LIN {X 0,Y 249.453,Z 553.415,A -85,B 0,C 180,E1 -18983.532,E2 -18983.532} C_VEL
LIN {X 0,Y 249.673,Z 553.384,A -85,B 0,C 180,E1 -18988.389,E2 -18988.389} C_VEL
LIN {X 0,Y 249.674,Z 553.383,A -85,B 0,C 180,E1 -18991.615,E2 -18991.615} C_VEL
LIN {X 0,Y 249.457,Z 553.406,A -85,B 0,C 180,E1 -18996.473,E2 -18996.473} C_VEL
LIN {X 0,Y 249.387,Z 553.419,A -85,B 0,C 180,E1 -18999.737,E2 -18999.737} C_VEL
LIN {X 0,Y 249.205,Z 553.438,A -85,B 0,C 180,E1 -19004.706,E2 -19004.706} C_VEL
LIN {X 0,Y 249.14,Z 553.449,A -85,B 0,C 180,E1 -19008.08,E2 -19008.08} C_VEL
LIN {X 0,Y 249.088,Z 553.442,A -85,B 0,C 180,E1 -19011.52,E2 -19011.52} C_VEL
LIN {X 0,Y 249.131,Z 553.45,A -85,B 0,C 180,E1 -19015.484,E2 -19015.484} C_VEL
LIN {X 0,Y 249.074,Z 553.461,A -85,B 0,C 180,E1 -19018.991,E2 -19018.991} C_VEL
LIN {X 0,Y 249.032,Z 553.458,A -85,B 0,C 180,E1 -19022.428,E2 -19022.428} C_VEL
LIN {X 0,Y 249.032,Z 553.463,A -85,B 0,C 180,E1 -19026.348,E2 -19026.348} C_VEL
LIN {X 0,Y 249.009,Z 553.46,A -85,B 0,C 180,E1 -19030.48,E2 -19030.48} C_VEL
LIN {X 0,Y 249.011,Z 553.466,A -85,B 0,C 180,E1 -19034.88,E2 -19034.88} C_VEL
LIN {X 0,Y 249.022,Z 553.465,A -85,B 0,C 180,E1 -19037.365,E2 -19037.365} C_VEL
LIN {X 0,Y 249.048,Z 553.457,A -85,B 0,C 180,E1 -19042.202,E2 -19042.202} C_VEL
LIN {X 0,Y 249.049,Z 553.463,A -85,B 0,C 180,E1 -19045.641,E2 -19045.641} C_VEL
LIN {X 0,Y 249.058,Z 553.456,A -85,B 0,C 180,E1 -19049.475,E2 -19049.475} C_VEL
LIN {X 0,Y 249.076,Z 553.452,A -85,B 0,C 180,E1 -19053.164,E2 -19053.164} C_VEL
LIN {X 0,Y 249.067,Z 553.458,A -85,B 0,C 180,E1 -19056.732,E2 -19056.732} C_VEL
LIN {X 0,Y 249.092,Z 553.451,A -85,B 0,C 180,E1 -19060.211,E2 -19060.211} C_VEL
LIN {X 0,Y 249.203,Z 553.435,A -85,B 0,C 180,E1 -19063.62,E2 -19063.62} C_VEL
LIN {X 0,Y 249.251,Z 553.435,A -85,B 0,C 180,E1 -19068.617,E2 -19068.617} C_VEL
LIN {X 0,Y 249.463,Z 553.405,A -85,B 0,C 180,E1 -19071.903,E2 -19071.903} C_VEL
LIN {X 0,Y 249.303,Z 553.423,A -85,B 0,C 180,E1 -19075.149,E2 -19075.149} C_VEL
LIN {X 0,Y 249.683,Z 553.382,A -85,B 0,C 180,E1 -19078.388,E2 -19078.388} C_VEL
LIN {X 0,Y 249.684,Z 553.383,A -85,B 0,C 180,E1 -19081.614,E2 -19081.614} C_VEL
LIN {X 0,Y 249.47,Z 553.408,A -85,B 0,C 180,E1 -19086.471,E2 -19086.471} C_VEL
LIN {X 0,Y 249.434,Z 553.416,A -85,B 0,C 180,E1 -19089.734,E2 -19089.734} C_VEL
LIN {X 0,Y 249.224,Z 553.432,A -85,B 0,C 180,E1 -19092.092,E2 -19092.092} C_VEL
LIN {X 0,Y 248.533,Z 553.52,A -85,B 0,C 180,E1 -19093.442,E2 -19093.442} C_VEL
LIN {X 0,Y 245.654,Z 553.884,A -85,B 0,C 180,E1 -19095.642,E2 -19095.642} C_VEL
LIN {X 0,Y 243.205,Z 554.19,A -85,B 0,C 180,E1 -19097.434,E2 -19097.434} C_VEL
LIN {X 0,Y 242.137,Z 554.321,A -85,B 0,C 180,E1 -19098.824,E2 -19098.824} C_VEL
LIN {X 0,Y 242.04,Z 554.328,A -85,B 0,C 180,E1 -19099.296,E2 -19099.296} C_VEL
LIN {X 0,Y 242.05,Z 554.315,A -85,B 0,C 180,E1 -19103.986,E2 -19103.986} C_VEL
LIN {X 0,Y 242.01,Z 554.334,A -85,B 0,C 180,E1 -19107.688,E2 -19107.688} C_VEL
LIN {X 0,Y 241.983,Z 554.34,A -85,B 0,C 180,E1 -19111.52,E2 -19111.52} C_VEL
LIN {X 0,Y 242.015,Z 554.338,A -85,B 0,C 180,E1 -19115.596,E2 -19115.596} C_VEL
LIN {X 0,Y 241.965,Z 554.344,A -85,B 0,C 180,E1 -19119.718,E2 -19119.718} C_VEL
LIN {X 0,Y 241.935,Z 554.349,A -85,B 0,C 180,E1 -19124.202,E2 -19124.202} C_VEL
LIN {X 0,Y 241.947,Z 554.347,A -85,B 0,C 180,E1 -19128.077,E2 -19128.077} C_VEL
LIN {X 0,Y 242.02,Z 554.338,A -85,B 0,C 180,E1 -19132.421,E2 -19132.421} C_VEL
LIN {X 0,Y 242.101,Z 554.421,A -85,B 0,C 180,E1 -19133.371,E2 -19133.371} C_VEL
LIN {X 0,Y 244.113,Z 564.051,A -85,B 0,C 180,E1 -19137.327,E2 -19137.327} C_VEL
LIN {X 0,Y 245.054,Z 568.388,A -85,B 0,C 180,E1 -19138.956,E2 -19138.956} C_VEL
LIN {X 0,Y 252.11,Z 587.582,A -85,B 0,C 180,E1 -19140.375,E2 -19140.375} C_VEL
LIN {X 0,Y 256.177,Z 617.752,A -85,B 0,C 180,E1 -19141.803,E2 -19141.803} C_VEL
LIN {X 0,Y 253.863,Z 677.446,A -85,B 0,C 180,E1 -19143.657,E2 -19143.657} C_VEL
LIN {X 0,Y 252.711,Z 691.266,A -85,B 0,C 180,E1 -19144.408,E2 -19144.408} C_VEL
LIN {X 0,Y 251.292,Z 703.771,A -85,B 0,C 180,E1 -19145.414,E2 -19145.414} C_VEL
LIN {X 0,Y 249.549,Z 716.207,A -85,B 0,C 180,E1 -19146.777,E2 -19146.777} C_VEL
LIN {X 0,Y 247.692,Z 727.365,A -85,B 0,C 180,E1 -19148.352,E2 -19148.352} C_VEL
LIN {X 0,Y 245.909,Z 737.764,A -85,B 0,C 180,E1 -19150.23,E2 -19150.23} C_VEL
LIN {X 0,Y 244.312,Z 747.422,A -85,B 0,C 180,E1 -19152.417,E2 -19152.417} C_VEL
LIN {X 0,Y 242.903,Z 754.812,A -85,B 0,C 180,E1 -19154.474,E2 -19154.474} C_VEL
LIN {X 0,Y 241.522,Z 762.054,A -85,B 0,C 180,E1 -19156.964,E2 -19156.964} C_VEL
LIN {X 0,Y 240.812,Z 766.949,A -85,B 0,C 180,E1 -19159.062,E2 -19159.062} C_VEL
LIN {X 0,Y 240.212,Z 771.663,A -85,B 0,C 180,E1 -19161.586,E2 -19161.586} C_VEL
LIN {X 0,Y 239.907,Z 775.221,A -85,B 0,C 180,E1 -19164.113,E2 -19164.113} C_VEL
LIN {X 0,Y 239.806,Z 777.727,A -85,B 0,C 180,E1 -19166.637,E2 -19166.637} C_VEL
LIN {X 0,Y 239.866,Z 778.859,A -85,B 0,C 180,E1 -19168.319,E2 -19168.319} C_VEL
LIN {X 0,Y 239.915,Z 779.546,A -85,B 0,C 180,E1 -19169.998,E2 -19169.998} C_VEL
LIN {X 0,Y 239.833,Z 779.83,A -85,B 0,C 180,E1 -19171.677,E2 -19171.677} C_VEL
LIN {X 0,Y 239.793,Z 779.295,A -85,B 0,C 180,E1 -19174.791,E2 -19174.791} C_VEL
LIN {X 0,Y 239.954,Z 778.232,A -85,B 0,C 180,E1 -19176.726,E2 -19176.726} C_VEL
LIN {X 0,Y 240.672,Z 775.128,A -85,B 0,C 180,E1 -19180.088,E2 -19180.088} C_VEL
LIN {X 0,Y 241.623,Z 771.637,A -85,B 0,C 180,E1 -19182.598,E2 -19182.598} C_VEL
LIN {X 0,Y 242.985,Z 767.08,A -85,B 0,C 180,E1 -19185.086,E2 -19185.086} C_VEL
LIN {X 0,Y 245.294,Z 760.216,A -85,B 0,C 180,E1 -19187.936,E2 -19187.936} C_VEL
LIN {X 0,Y 247.599,Z 752.325,A -85,B 0,C 180,E1 -19190.495,E2 -19190.495} C_VEL
LIN {X 0,Y 250.22,Z 743.627,A -85,B 0,C 180,E1 -19192.716,E2 -19192.716} C_VEL
LIN {X 0,Y 253.211,Z 733.103,A -85,B 0,C 180,E1 -19194.819,E2 -19194.819} C_VEL
LIN {X 0,Y 255.815,Z 722.508,A -85,B 0,C 180,E1 -19196.512,E2 -19196.512} C_VEL
LIN {X 0,Y 258.523,Z 710.623,A -85,B 0,C 180,E1 -19197.963,E2 -19197.963} C_VEL
LIN {X 0,Y 260.759,Z 698.126,A -85,B 0,C 180,E1 -19199.129,E2 -19199.129} C_VEL
LIN {X 0,Y 262.607,Z 685.023,A -85,B 0,C 180,E1 -19200.005,E2 -19200.005} C_VEL
LIN {X 0,Y 263.954,Z 670.854,A -85,B 0,C 180,E1 -19200.603,E2 -19200.603} C_VEL
LIN {X 0,Y 266.576,Z 619.411,A -85,B 0,C 180,E1 -19202.173,E2 -19202.173} C_VEL
LIN {X 0,Y 264.465,Z 603.384,A -85,B 0,C 180,E1 -19203.2,E2 -19203.2} C_VEL
LIN {X 0,Y 260.104,Z 593.001,A -85,B 0,C 180,E1 -19204.48,E2 -19204.48} C_VEL
LIN {X 0,Y 253.772,Z 580.509,A -85,B 0,C 180,E1 -19206.375,E2 -19206.375} C_VEL
LIN {X 0,Y 250.696,Z 575.081,A -85,B 0,C 180,E1 -19207.34,E2 -19207.34} C_VEL
LIN {X 0,Y 247.979,Z 570.475,A -85,B 0,C 180,E1 -19208.225,E2 -19208.225} C_VEL
LIN {X 0,Y 245.387,Z 565.842,A -85,B 0,C 180,E1 -19209.17,E2 -19209.17} C_VEL
LIN {X 0,Y 243.644,Z 560.104,A -85,B 0,C 180,E1 -19212.645,E2 -19212.645} C_VEL
LIN {X 0,Y 241.944,Z 554.347,A -85,B 0,C 180,E1 -19216.7,E2 -19216.7} C_VEL
LIN {X 0,Y 241.975,Z 554.339,A -85,B 0,C 180,E1 -19220.284,E2 -19220.284} C_VEL
LIN {X 0,Y 242.03,Z 554.338,A -85,B 0,C 180,E1 -19224.495,E2 -19224.495} C_VEL
LIN {X 0,Y 241.968,Z 554.338,A -85,B 0,C 180,E1 -19228.478,E2 -19228.478} C_VEL
LIN {X 0,Y 242,Z 554.332,A -85,B 0,C 180,E1 -19232.311,E2 -19232.311} C_VEL
LIN {X 0,Y 242.049,Z 554.325,A -85,B 0,C 180,E1 -19236.014,E2 -19236.014} C_VEL
LIN {X 0,Y 242.028,Z 554.328,A -85,B 0,C 180,E1 -19239.606,E2 -19239.606} C_VEL
LIN {X 0,Y 242.154,Z 554.315,A -85,B 0,C 180,E1 -19243.277,E2 -19243.277} C_VEL
LIN {X 0,Y 242.177,Z 554.308,A -85,B 0,C 180,E1 -19248.278,E2 -19248.278} C_VEL
LIN {X 0,Y 242.425,Z 554.278,A -85,B 0,C 180,E1 -19251.665,E2 -19251.665} C_VEL
LIN {X 0,Y 242.252,Z 554.301,A -85,B 0,C 180,E1 -19255.006,E2 -19255.006} C_VEL
LIN {X 0,Y 242.629,Z 554.255,A -85,B 0,C 180,E1 -19258.339,E2 -19258.339} C_VEL
LIN {X 0,Y 242.634,Z 554.256,A -85,B 0,C 180,E1 -19261.659,E2 -19261.659} C_VEL
LIN {X 0,Y 242.427,Z 554.334,A -85,B 0,C 180,E1 -19267.914,E2 -19267.914} C_VEL
LIN {X 0,Y 243.227,Z 557.795,A -85,B 0,C 180,E1 -19270.351,E2 -19270.351} C_VEL
LIN {X 0,Y 245.42,Z 561.512,A -85,B 0,C 180,E1 -19271.144,E2 -19271.144} C_VEL
LIN {X 0,Y 247.197,Z 563.941,A -85,B 0,C 180,E1 -19271.738,E2 -19271.738} C_VEL
LIN {X 0,Y 250.763,Z 569.544,A -85,B 0,C 180,E1 -19272.904,E2 -19272.904} C_VEL
LIN {X 0,Y 255.426,Z 577.254,A -85,B 0,C 180,E1 -19274.337,E2 -19274.337} C_VEL
LIN {X 0,Y 260.585,Z 586.905,A -85,B 0,C 180,E1 -19275.848,E2 -19275.848} C_VEL
LIN {X 0,Y 265.939,Z 598.808,A -85,B 0,C 180,E1 -19277.377,E2 -19277.377} C_VEL
LIN {X 0,Y 267.443,Z 602.427,A -85,B 0,C 180,E1 -19277.8,E2 -19277.8} C_VEL
LIN {X 0,Y 263.978,Z 664.442,A -85,B 0,C 180,E1 -19279.693,E2 -19279.693} C_VEL
LIN {X 0,Y 262.673,Z 677.208,A -85,B 0,C 180,E1 -19280.353,E2 -19280.353} C_VEL
LIN {X 0,Y 260.893,Z 690.002,A -85,B 0,C 180,E1 -19281.324,E2 -19281.324} C_VEL
LIN {X 0,Y 258.594,Z 702.502,A -85,B 0,C 180,E1 -19282.627,E2 -19282.627} C_VEL
LIN {X 0,Y 256.222,Z 713.303,A -85,B 0,C 180,E1 -19284.087,E2 -19284.087} C_VEL
LIN {X 0,Y 253.528,Z 724.026,A -85,B 0,C 180,E1 -19285.934,E2 -19285.934} C_VEL
LIN {X 0,Y 250.699,Z 733.84,A -85,B 0,C 180,E1 -19288.081,E2 -19288.081} C_VEL
LIN {X 0,Y 248.21,Z 741.845,A -85,B 0,C 180,E1 -19290.272,E2 -19290.272} C_VEL
LIN {X 0,Y 246.081,Z 748.371,A -85,B 0,C 180,E1 -19292.505,E2 -19292.505} C_VEL
LIN {X 0,Y 243.964,Z 754.493,A -85,B 0,C 180,E1 -19295.179,E2 -19295.179} C_VEL
LIN {X 0,Y 242.565,Z 758.575,A -85,B 0,C 180,E1 -19297.476,E2 -19297.476} C_VEL
LIN {X 0,Y 241.136,Z 762.726,A -85,B 0,C 180,E1 -19300.735,E2 -19300.735} C_VEL
LIN {X 0,Y 240.385,Z 764.662,A -85,B 0,C 180,E1 -19303.041,E2 -19303.041} C_VEL
LIN {X 0,Y 239.891,Z 765.829,A -85,B 0,C 180,E1 -19305.326,E2 -19305.326} C_VEL
LIN {X 0,Y 239.58,Z 766.222,A -85,B 0,C 180,E1 -19307.573,E2 -19307.573} C_VEL
LIN {X 0,Y 239.453,Z 765.906,A -85,B 0,C 180,E1 -19309.785,E2 -19309.785} C_VEL
LIN {X 0,Y 239.507,Z 764.641,A -85,B 0,C 180,E1 -19312.397,E2 -19312.397} C_VEL
LIN {X 0,Y 239.812,Z 762.222,A -85,B 0,C 180,E1 -19315.141,E2 -19315.141} C_VEL
LIN {X 0,Y 240.468,Z 758.038,A -85,B 0,C 180,E1 -19318.263,E2 -19318.263} C_VEL
LIN {X 0,Y 241.28,Z 753.121,A -85,B 0,C 180,E1 -19320.906,E2 -19320.906} C_VEL
LIN {X 0,Y 242.421,Z 746.61,A -85,B 0,C 180,E1 -19323.596,E2 -19323.596} C_VEL
LIN {X 0,Y 243.952,Z 738.534,A -85,B 0,C 180,E1 -19326.217,E2 -19326.217} C_VEL
LIN {X 0,Y 245.532,Z 730.166,A -85,B 0,C 180,E1 -19328.378,E2 -19328.378} C_VEL
LIN {X 0,Y 247.276,Z 719.954,A -85,B 0,C 180,E1 -19330.494,E2 -19330.494} C_VEL
LIN {X 0,Y 249.194,Z 708.613,A -85,B 0,C 180,E1 -19332.351,E2 -19332.351} C_VEL
LIN {X 0,Y 250.796,Z 696.998,A -85,B 0,C 180,E1 -19333.833,E2 -19333.833} C_VEL
LIN {X 0,Y 252.352,Z 684.2,A -85,B 0,C 180,E1 -19335.074,E2 -19335.074} C_VEL
LIN {X 0,Y 253.441,Z 671.386,A -85,B 0,C 180,E1 -19335.968,E2 -19335.968} C_VEL
LIN {X 0,Y 254.324,Z 657.187,A -85,B 0,C 180,E1 -19336.593,E2 -19336.593} C_VEL
LIN {X 0,Y 256.812,Z 593.445,A -85,B 0,C 180,E1 -19338.515,E2 -19338.515} C_VEL
LIN {X 0,Y 249.263,Z 572.337,A -85,B 0,C 180,E1 -19340.004,E2 -19340.004} C_VEL
LIN {X 0,Y 242.612,Z 555.291,A -85,B 0,C 180,E1 -19341.36,E2 -19341.36} C_VEL
LIN {X 0,Y 242.438,Z 554.287,A -85,B 0,C 180,E1 -19341.878,E2 -19341.878} C_VEL
LIN {X 0,Y 242.372,Z 554.299,A -85,B 0,C 180,E1 -19346.678,E2 -19346.678} C_VEL
LIN {X 0,Y 242.634,Z 554.261,A -85,B 0,C 180,E1 -19348.343,E2 -19348.343} C_VEL
LIN {X 0,Y 242.634,Z 554.259,A -85,B 0,C 180,E1 -19351.662,E2 -19351.662} C_VEL
LIN {X 0,Y 242.43,Z 554.282,A -85,B 0,C 180,E1 -19356.661,E2 -19356.661} C_VEL
LIN {X 0,Y 242.313,Z 554.3,A -85,B 0,C 180,E1 -19360.024,E2 -19360.024} C_VEL
LIN {X 0,Y 242.166,Z 554.318,A -85,B 0,C 180,E1 -19365.143,E2 -19365.143} C_VEL
LIN {X 0,Y 242.073,Z 554.33,A -85,B 0,C 180,E1 -19368.626,E2 -19368.626} C_VEL
LIN {X 0,Y 242.014,Z 554.32,A -85,B 0,C 180,E1 -19372.182,E2 -19372.182} C_VEL
LIN {X 0,Y 242.068,Z 554.329,A -85,B 0,C 180,E1 -19375.84,E2 -19375.84} C_VEL
LIN {X 0,Y 242.009,Z 554.339,A -85,B 0,C 180,E1 -19379.586,E2 -19379.586} C_VEL
LIN {X 0,Y 241.983,Z 554.342,A -85,B 0,C 180,E1 -19383.495,E2 -19383.495} C_VEL
LIN {X 0,Y 241.989,Z 554.341,A -85,B 0,C 180,E1 -19387.585,E2 -19387.585} C_VEL
LIN {X 0,Y 241.942,Z 554.343,A -85,B 0,C 180,E1 -19391.924,E2 -19391.924} C_VEL
LIN {X 0,Y 241.941,Z 554.346,A -85,B 0,C 180,E1 -19396.573,E2 -19396.573} C_VEL
LIN {X 0,Y 241.961,Z 554.333,A -85,B 0,C 180,E1 -19400.283,E2 -19400.283} C_VEL
LIN {X 0,Y 241.992,Z 554.339,A -85,B 0,C 180,E1 -19404.491,E2 -19404.491} C_VEL
LIN {X 0,Y 241.98,Z 554.338,A -85,B 0,C 180,E1 -19408.482,E2 -19408.482} C_VEL
LIN {X 0,Y 242.013,Z 554.33,A -85,B 0,C 180,E1 -19412.314,E2 -19412.314} C_VEL
LIN {X 0,Y 242.047,Z 554.333,A -85,B 0,C 180,E1 -19416.016,E2 -19416.016} C_VEL
LIN {X 0,Y 242.028,Z 554.334,A -85,B 0,C 180,E1 -19419.608,E2 -19419.608} C_VEL
LIN {X 0,Y 242.134,Z 554.312,A -85,B 0,C 180,E1 -19423.308,E2 -19423.308} C_VEL
LIN {X 0,Y 242.186,Z 554.315,A -85,B 0,C 180,E1 -19428.281,E2 -19428.281} C_VEL
LIN {X 0,Y 242.409,Z 554.285,A -85,B 0,C 180,E1 -19431.666,E2 -19431.666} C_VEL
LIN {X 0,Y 242.263,Z 554.299,A -85,B 0,C 180,E1 -19435.008,E2 -19435.008} C_VEL
LIN {X 0,Y 242.644,Z 554.259,A -85,B 0,C 180,E1 -19438.341,E2 -19438.341} C_VEL
LIN {X 0,Y 242.644,Z 554.259,A -85,B 0,C 180,E1 -19441.661,E2 -19441.661} C_VEL
LIN {X 0,Y 242.443,Z 554.282,A -85,B 0,C 180,E1 -19446.659,E2 -19446.659} C_VEL
LIN {X 0,Y 242.355,Z 554.296,A -85,B 0,C 180,E1 -19450.021,E2 -19450.021} C_VEL
LIN {X 0,Y 242.176,Z 554.315,A -85,B 0,C 180,E1 -19455.141,E2 -19455.141} C_VEL
LIN {X 0,Y 242.04,Z 554.328,A -85,B 0,C 180,E1 -19459.296,E2 -19459.296} C_VEL
LIN {X 0,Y 241.363,Z 554.413,A -85,B 0,C 180,E1 -19460.683,E2 -19460.683} C_VEL
LIN {X 0,Y 238.564,Z 554.765,A -85,B 0,C 180,E1 -19462.948,E2 -19462.948} C_VEL
LIN {X 0,Y 235.339,Z 555.168,A -85,B 0,C 180,E1 -19465.741,E2 -19465.741} C_VEL
LIN {X 0,Y 234.973,Z 555.209,A -85,B 0,C 180,E1 -19466.707,E2 -19466.707} C_VEL
LIN {X 0,Y 234.932,Z 555.22,A -85,B 0,C 180,E1 -19470.569,E2 -19470.569} C_VEL
LIN {X 0,Y 234.951,Z 555.219,A -85,B 0,C 180,E1 -19474.635,E2 -19474.635} C_VEL
LIN {X 0,Y 234.951,Z 555.217,A -85,B 0,C 180,E1 -19478.944,E2 -19478.944} C_VEL
LIN {X 0,Y 234.894,Z 555.225,A -85,B 0,C 180,E1 -19483.486,E2 -19483.486} C_VEL
LIN {X 0,Y 234.889,Z 555.225,A -85,B 0,C 180,E1 -19486.511,E2 -19486.511} C_VEL
LIN {X 0,Y 234.964,Z 555.215,A -85,B 0,C 180,E1 -19491.085,E2 -19491.085} C_VEL
LIN {X 0,Y 235.002,Z 555.272,A -85,B 0,C 180,E1 -19492.793,E2 -19492.793} C_VEL
LIN {X 0,Y 236.752,Z 563.305,A -85,B 0,C 180,E1 -19496.222,E2 -19496.222} C_VEL
LIN {X 0,Y 237.673,Z 567.846,A -85,B 0,C 180,E1 -19498.087,E2 -19498.087} C_VEL
LIN {X 0,Y 245.755,Z 589.508,A -85,B 0,C 180,E1 -19499.791,E2 -19499.791} C_VEL
LIN {X 0,Y 249.596,Z 618.208,A -85,B 0,C 180,E1 -19501.197,E2 -19501.197} C_VEL
LIN {X 0,Y 247.233,Z 676.781,A -85,B 0,C 180,E1 -19503.058,E2 -19503.058} C_VEL
LIN {X 0,Y 246.068,Z 690.839,A -85,B 0,C 180,E1 -19503.835,E2 -19503.835} C_VEL
LIN {X 0,Y 244.622,Z 702.904,A -85,B 0,C 180,E1 -19504.811,E2 -19504.811} C_VEL
LIN {X 0,Y 242.966,Z 714.687,A -85,B 0,C 180,E1 -19506.109,E2 -19506.109} C_VEL
LIN {X 0,Y 241.115,Z 726.104,A -85,B 0,C 180,E1 -19507.731,E2 -19507.731} C_VEL
LIN {X 0,Y 239.265,Z 736.522,A -85,B 0,C 180,E1 -19509.606,E2 -19509.606} C_VEL
LIN {X 0,Y 237.742,Z 744.873,A -85,B 0,C 180,E1 -19511.469,E2 -19511.469} C_VEL
LIN {X 0,Y 236.218,Z 752.657,A -85,B 0,C 180,E1 -19513.579,E2 -19513.579} C_VEL
LIN {X 0,Y 234.769,Z 760.268,A -85,B 0,C 180,E1 -19516.141,E2 -19516.141} C_VEL
LIN {X 0,Y 233.802,Z 766.371,A -85,B 0,C 180,E1 -19518.73,E2 -19518.73} C_VEL
LIN {X 0,Y 233.178,Z 771.168,A -85,B 0,C 180,E1 -19521.33,E2 -19521.33} C_VEL
LIN {X 0,Y 232.832,Z 774.8,A -85,B 0,C 180,E1 -19523.933,E2 -19523.933} C_VEL
LIN {X 0,Y 232.714,Z 777.374,A -85,B 0,C 180,E1 -19526.535,E2 -19526.535} C_VEL
LIN {X 0,Y 232.776,Z 778.565,A -85,B 0,C 180,E1 -19528.267,E2 -19528.267} C_VEL
LIN {X 0,Y 232.846,Z 779.292,A -85,B 0,C 180,E1 -19529.998,E2 -19529.998} C_VEL
LIN {X 0,Y 232.745,Z 779.606,A -85,B 0,C 180,E1 -19531.728,E2 -19531.728} C_VEL
LIN {X 0,Y 232.709,Z 779.21,A -85,B 0,C 180,E1 -19534.7,E2 -19534.7} C_VEL
LIN {X 0,Y 232.892,Z 778.141,A -85,B 0,C 180,E1 -19536.93,E2 -19536.93} C_VEL
LIN {X 0,Y 233.67,Z 775.113,A -85,B 0,C 180,E1 -19540.394,E2 -19540.394} C_VEL
LIN {X 0,Y 234.659,Z 771.696,A -85,B 0,C 180,E1 -19542.978,E2 -19542.978} C_VEL
LIN {X 0,Y 236.144,Z 767.215,A -85,B 0,C 180,E1 -19545.534,E2 -19545.534} C_VEL
LIN {X 0,Y 238.188,Z 761.546,A -85,B 0,C 180,E1 -19548.045,E2 -19548.045} C_VEL
LIN {X 0,Y 240.41,Z 754.539,A -85,B 0,C 180,E1 -19550.534,E2 -19550.534} C_VEL
LIN {X 0,Y 243.215,Z 745.813,A -85,B 0,C 180,E1 -19552.958,E2 -19552.958} C_VEL
LIN {X 0,Y 245.94,Z 736.924,A -85,B 0,C 180,E1 -19554.926,E2 -19554.926} C_VEL
LIN {X 0,Y 248.95,Z 726.04,A -85,B 0,C 180,E1 -19556.849,E2 -19556.849} C_VEL
LIN {X 0,Y 251.617,Z 715.119,A -85,B 0,C 180,E1 -19558.346,E2 -19558.346} C_VEL
LIN {X 0,Y 254.084,Z 703.044,A -85,B 0,C 180,E1 -19559.629,E2 -19559.629} C_VEL
LIN {X 0,Y 256.216,Z 690.498,A -85,B 0,C 180,E1 -19560.606,E2 -19560.606} C_VEL
LIN {X 0,Y 257.82,Z 677.589,A -85,B 0,C 180,E1 -19561.29,E2 -19561.29} C_VEL
LIN {X 0,Y 259.171,Z 655.609,A -85,B 0,C 180,E1 -19562.037,E2 -19562.037} C_VEL
LIN {X 0,Y 261.121,Z 620.828,A -85,B 0,C 180,E1 -19563.109,E2 -19563.109} C_VEL
LIN {X 0,Y 259.252,Z 606.142,A -85,B 0,C 180,E1 -19564.087,E2 -19564.087} C_VEL
LIN {X 0,Y 255.41,Z 597.072,A -85,B 0,C 180,E1 -19565.262,E2 -19565.262} C_VEL
LIN {X 0,Y 249.588,Z 585.241,A -85,B 0,C 180,E1 -19567.122,E2 -19567.122} C_VEL
LIN {X 0,Y 244.593,Z 576.151,A -85,B 0,C 180,E1 -19568.816,E2 -19568.816} C_VEL
LIN {X 0,Y 241.799,Z 571.478,A -85,B 0,C 180,E1 -19569.816,E2 -19569.816} C_VEL
LIN {X 0,Y 238.536,Z 566.681,A -85,B 0,C 180,E1 -19571.014,E2 -19571.014} C_VEL
LIN {X 0,Y 238.014,Z 565.519,A -85,B 0,C 180,E1 -19571.262,E2 -19571.262} C_VEL
LIN {X 0,Y 236.021,Z 559.128,A -85,B 0,C 180,E1 -19575.61,E2 -19575.61} C_VEL
LIN {X 0,Y 234.914,Z 555.224,A -85,B 0,C 180,E1 -19578.695,E2 -19578.695} C_VEL
LIN {X 0,Y 234.949,Z 555.22,A -85,B 0,C 180,E1 -19581.084,E2 -19581.084} C_VEL
LIN {X 0,Y 234.954,Z 555.211,A -85,B 0,C 180,E1 -19585.365,E2 -19585.365} C_VEL
LIN {X 0,Y 234.962,Z 555.212,A -85,B 0,C 180,E1 -19590.155,E2 -19590.155} C_VEL
LIN {X 0,Y 234.986,Z 555.208,A -85,B 0,C 180,E1 -19593.792,E2 -19593.792} C_VEL
LIN {X 0,Y 235.002,Z 555.21,A -85,B 0,C 180,E1 -19598.968,E2 -19598.968} C_VEL
LIN {X 0,Y 235.087,Z 555.197,A -85,B 0,C 180,E1 -19603.058,E2 -19603.058} C_VEL
LIN {X 0,Y 235.137,Z 555.185,A -85,B 0,C 180,E1 -19607.922,E2 -19607.922} C_VEL
LIN {X 0,Y 235.38,Z 555.156,A -85,B 0,C 180,E1 -19611.413,E2 -19611.413} C_VEL
LIN {X 0,Y 235.396,Z 555.16,A -85,B 0,C 180,E1 -19613.14,E2 -19613.14} C_VEL
LIN {X 0,Y 235.589,Z 555.132,A -85,B 0,C 180,E1 -19618.29,E2 -19618.29} C_VEL
LIN {X 0,Y 235.594,Z 555.132,A -85,B 0,C 180,E1 -19621.709,E2 -19621.709} C_VEL
LIN {X 0,Y 235.329,Z 555.373,A -85,B 0,C 180,E1 -19625.999,E2 -19625.999} C_VEL
LIN {X 0,Y 236.231,Z 558.24,A -85,B 0,C 180,E1 -19628.285,E2 -19628.285} C_VEL
LIN {X 0,Y 238.933,Z 562.454,A -85,B 0,C 180,E1 -19629.363,E2 -19629.363} C_VEL
LIN {X 0,Y 240.45,Z 564.773,A -85,B 0,C 180,E1 -19629.94,E2 -19629.94} C_VEL
LIN {X 0,Y 243.748,Z 569.674,A -85,B 0,C 180,E1 -19631.117,E2 -19631.117} C_VEL
LIN {X 0,Y 248.598,Z 577.378,A -85,B 0,C 180,E1 -19632.759,E2 -19632.759} C_VEL
LIN {X 0,Y 254.741,Z 588.537,A -85,B 0,C 180,E1 -19634.698,E2 -19634.698} C_VEL
LIN {X 0,Y 260.224,Z 600.408,A -85,B 0,C 180,E1 -19636.351,E2 -19636.351} C_VEL
LIN {X 0,Y 261.908,Z 604.641,A -85,B 0,C 180,E1 -19636.856,E2 -19636.856} C_VEL
LIN {X 0,Y 258.357,Z 664.938,A -85,B 0,C 180,E1 -19638.753,E2 -19638.753} C_VEL
LIN {X 0,Y 256.962,Z 677.702,A -85,B 0,C 180,E1 -19639.429,E2 -19639.429} C_VEL
LIN {X 0,Y 255.025,Z 690.841,A -85,B 0,C 180,E1 -19640.459,E2 -19640.459} C_VEL
LIN {X 0,Y 252.711,Z 702.778,A -85,B 0,C 180,E1 -19641.729,E2 -19641.729} C_VEL
LIN {X 0,Y 250.377,Z 713.056,A -85,B 0,C 180,E1 -19643.139,E2 -19643.139} C_VEL
LIN {X 0,Y 247.64,Z 723.57,A -85,B 0,C 180,E1 -19644.954,E2 -19644.954} C_VEL
LIN {X 0,Y 244.692,Z 733.29,A -85,B 0,C 180,E1 -19647.086,E2 -19647.086} C_VEL
LIN {X 0,Y 241.67,Z 742.413,A -85,B 0,C 180,E1 -19649.628,E2 -19649.628} C_VEL
LIN {X 0,Y 238.959,Z 750.102,A -85,B 0,C 180,E1 -19652.438,E2 -19652.438} C_VEL
LIN {X 0,Y 236.707,Z 756.185,A -85,B 0,C 180,E1 -19655.34,E2 -19655.34} C_VEL
LIN {X 0,Y 235.309,Z 759.946,A -85,B 0,C 180,E1 -19657.722,E2 -19657.722} C_VEL
LIN {X 0,Y 234.252,Z 762.805,A -85,B 0,C 180,E1 -19660.132,E2 -19660.132} C_VEL
LIN {X 0,Y 233.134,Z 765.483,A -85,B 0,C 180,E1 -19663.66,E2 -19663.66} C_VEL
LIN {X 0,Y 232.595,Z 766.378,A -85,B 0,C 180,E1 -19666.482,E2 -19666.482} C_VEL
LIN {X 0,Y 232.349,Z 766.261,A -85,B 0,C 180,E1 -19669.128,E2 -19669.128} C_VEL
LIN {X 0,Y 232.368,Z 765.154,A -85,B 0,C 180,E1 -19671.846,E2 -19671.846} C_VEL
LIN {X 0,Y 232.701,Z 762.58,A -85,B 0,C 180,E1 -19674.985,E2 -19674.985} C_VEL
LIN {X 0,Y 233.216,Z 759.429,A -85,B 0,C 180,E1 -19677.54,E2 -19677.54} C_VEL
LIN {X 0,Y 234.023,Z 754.315,A -85,B 0,C 180,E1 -19680.562,E2 -19680.562} C_VEL
LIN {X 0,Y 235.184,Z 748.033,A -85,B 0,C 180,E1 -19683.372,E2 -19683.372} C_VEL
LIN {X 0,Y 236.719,Z 740.027,A -85,B 0,C 180,E1 -19686.132,E2 -19686.132} C_VEL
LIN {X 0,Y 238.496,Z 730.928,A -85,B 0,C 180,E1 -19688.616,E2 -19688.616} C_VEL
LIN {X 0,Y 240.329,Z 720.712,A -85,B 0,C 180,E1 -19690.814,E2 -19690.814} C_VEL
LIN {X 0,Y 242.21,Z 710.041,A -85,B 0,C 180,E1 -19692.638,E2 -19692.638} C_VEL
LIN {X 0,Y 243.81,Z 699.249,A -85,B 0,C 180,E1 -19694.109,E2 -19694.109} C_VEL
LIN {X 0,Y 245.309,Z 687.622,A -85,B 0,C 180,E1 -19695.332,E2 -19695.332} C_VEL
LIN {X 0,Y 246.541,Z 674.504,A -85,B 0,C 180,E1 -19696.357,E2 -19696.357} C_VEL
LIN {X 0,Y 247.514,Z 661.487,A -85,B 0,C 180,E1 -19697.029,E2 -19697.029} C_VEL
LIN {X 0,Y 250.202,Z 594.692,A -85,B 0,C 180,E1 -19699.119,E2 -19699.119} C_VEL
LIN {X 0,Y 242.479,Z 573.311,A -85,B 0,C 180,E1 -19700.693,E2 -19700.693} C_VEL
LIN {X 0,Y 235.45,Z 555.519,A -85,B 0,C 180,E1 -19702.175,E2 -19702.175} C_VEL
LIN {X 0,Y 235.354,Z 555.17,A -85,B 0,C 180,E1 -19702.496,E2 -19702.496} C_VEL
LIN {X 0,Y 235.594,Z 555.138,A -85,B 0,C 180,E1 -19708.293,E2 -19708.293} C_VEL
LIN {X 0,Y 235.594,Z 555.136,A -85,B 0,C 180,E1 -19711.712,E2 -19711.712} C_VEL
LIN {X 0,Y 235.401,Z 555.159,A -85,B 0,C 180,E1 -19716.861,E2 -19716.861} C_VEL
LIN {X 0,Y 235.237,Z 555.182,A -85,B 0,C 180,E1 -19720.329,E2 -19720.329} C_VEL
LIN {X 0,Y 235.113,Z 555.197,A -85,B 0,C 180,E1 -19725.609,E2 -19725.609} C_VEL
LIN {X 0,Y 235.009,Z 555.207,A -85,B 0,C 180,E1 -19729.208,E2 -19729.208} C_VEL
LIN {X 0,Y 234.962,Z 555.199,A -85,B 0,C 180,E1 -19732.885,E2 -19732.885} C_VEL
LIN {X 0,Y 234.969,Z 555.213,A -85,B 0,C 180,E1 -19736.66,E2 -19736.66} C_VEL
LIN {X 0,Y 234.924,Z 555.22,A -85,B 0,C 180,E1 -19740.571,E2 -19740.571} C_VEL
LIN {X 0,Y 234.929,Z 555.219,A -85,B 0,C 180,E1 -19744.641,E2 -19744.641} C_VEL
LIN {X 0,Y 234.945,Z 555.218,A -85,B 0,C 180,E1 -19748.947,E2 -19748.947} C_VEL
LIN {X 0,Y 234.893,Z 555.226,A -85,B 0,C 180,E1 -19753.488,E2 -19753.488} C_VEL
LIN {X 0,Y 234.894,Z 555.223,A -85,B 0,C 180,E1 -19756.517,E2 -19756.517} C_VEL
LIN {X 0,Y 234.922,Z 555.211,A -85,B 0,C 180,E1 -19761.081,E2 -19761.081} C_VEL
LIN {X 0,Y 234.935,Z 555.221,A -85,B 0,C 180,E1 -19765.364,E2 -19765.364} C_VEL
LIN {X 0,Y 234.937,Z 555.214,A -85,B 0,C 180,E1 -19769.434,E2 -19769.434} C_VEL
LIN {X 0,Y 235.001,Z 555.209,A -85,B 0,C 180,E1 -19773.796,E2 -19773.796} C_VEL
LIN {X 0,Y 234.997,Z 555.21,A -85,B 0,C 180,E1 -19778.969,E2 -19778.969} C_VEL
LIN {X 0,Y 235.071,Z 555.19,A -85,B 0,C 180,E1 -19783.088,E2 -19783.088} C_VEL
LIN {X 0,Y 235.118,Z 555.198,A -85,B 0,C 180,E1 -19787.923,E2 -19787.923} C_VEL
LIN {X 0,Y 235.34,Z 555.167,A -85,B 0,C 180,E1 -19791.414,E2 -19791.414} C_VEL
LIN {X 0,Y 235.382,Z 555.155,A -85,B 0,C 180,E1 -19793.142,E2 -19793.142} C_VEL
LIN {X 0,Y 235.604,Z 555.136,A -85,B 0,C 180,E1 -19798.292,E2 -19798.292} C_VEL
LIN {X 0,Y 235.604,Z 555.135,A -85,B 0,C 180,E1 -19801.71,E2 -19801.71} C_VEL
LIN {X 0,Y 235.415,Z 555.158,A -85,B 0,C 180,E1 -19806.859,E2 -19806.859} C_VEL
LIN {X 0,Y 235.263,Z 555.177,A -85,B 0,C 180,E1 -19810.326,E2 -19810.326} C_VEL
LIN {X 0,Y 235.123,Z 555.196,A -85,B 0,C 180,E1 -19815.607,E2 -19815.607} C_VEL
LIN {X 0,Y 235.012,Z 555.208,A -85,B 0,C 180,E1 -19819.269,E2 -19819.269} C_VEL
LIN {X 0,Y 234.962,Z 555.198,A -85,B 0,C 180,E1 -19822.884,E2 -19822.884} C_VEL
LIN {X 0,Y 234.973,Z 555.209,A -85,B 0,C 180,E1 -19826.707,E2 -19826.707} C_VEL
LIN {X 0,Y 234.236,Z 555.305,A -85,B 0,C 180,E1 -19828.137,E2 -19828.137} C_VEL
LIN {X 0,Y 231.379,Z 555.663,A -85,B 0,C 180,E1 -19830.473,E2 -19830.473} C_VEL
LIN {X 0,Y 228.986,Z 555.962,A -85,B 0,C 180,E1 -19832.376,E2 -19832.376} C_VEL
LIN {X 0,Y 227.95,Z 556.091,A -85,B 0,C 180,E1 -19833.853,E2 -19833.853} C_VEL
LIN {X 0,Y 227.858,Z 556.098,A -85,B 0,C 180,E1 -19834.353,E2 -19834.353} C_VEL
LIN {X 0,Y 227.853,Z 556.106,A -85,B 0,C 180,E1 -19838.09,E2 -19838.09} C_VEL
LIN {X 0,Y 227.819,Z 556.107,A -85,B 0,C 180,E1 -19842.742,E2 -19842.742} C_VEL
LIN {X 0,Y 227.818,Z 556.107,A -85,B 0,C 180,E1 -19847.256,E2 -19847.256} C_VEL
LIN {X 0,Y 227.951,Z 556.123,A -85,B 0,C 180,E1 -19852.191,E2 -19852.191} C_VEL
LIN {X 0,Y 229.829,Z 564.734,A -85,B 0,C 180,E1 -19855.99,E2 -19855.99} C_VEL
LIN {X 0,Y 230.438,Z 567.752,A -85,B 0,C 180,E1 -19857.257,E2 -19857.257} C_VEL
LIN {X 0,Y 239.392,Z 591.57,A -85,B 0,C 180,E1 -19859.188,E2 -19859.188} C_VEL
LIN {X 0,Y 243.017,Z 618.467,A -85,B 0,C 180,E1 -19860.549,E2 -19860.549} C_VEL
LIN {X 0,Y 240.656,Z 676.267,A -85,B 0,C 180,E1 -19862.437,E2 -19862.437} C_VEL
LIN {X 0,Y 239.499,Z 689.647,A -85,B 0,C 180,E1 -19863.179,E2 -19863.179} C_VEL
LIN {X 0,Y 238.008,Z 701.979,A -85,B 0,C 180,E1 -19864.178,E2 -19864.178} C_VEL
LIN {X 0,Y 236.437,Z 713.154,A -85,B 0,C 180,E1 -19865.406,E2 -19865.406} C_VEL
LIN {X 0,Y 234.573,Z 724.82,A -85,B 0,C 180,E1 -19867.075,E2 -19867.075} C_VEL
LIN {X 0,Y 232.778,Z 734.247,A -85,B 0,C 180,E1 -19868.756,E2 -19868.756} C_VEL
LIN {X 0,Y 230.972,Z 743.475,A -85,B 0,C 180,E1 -19870.787,E2 -19870.787} C_VEL
LIN {X 0,Y 229.693,Z 750.38,A -85,B 0,C 180,E1 -19872.641,E2 -19872.641} C_VEL
LIN {X 0,Y 228.113,Z 758.445,A -85,B 0,C 180,E1 -19875.273,E2 -19875.273} C_VEL
LIN {X 0,Y 227.073,Z 763.883,A -85,B 0,C 180,E1 -19877.485,E2 -19877.485} C_VEL
LIN {X 0,Y 226.32,Z 769.192,A -85,B 0,C 180,E1 -19880.164,E2 -19880.164} C_VEL
LIN {X 0,Y 225.839,Z 773.274,A -85,B 0,C 180,E1 -19882.847,E2 -19882.847} C_VEL
LIN {X 0,Y 225.638,Z 776.093,A -85,B 0,C 180,E1 -19885.361,E2 -19885.361} C_VEL
LIN {X 0,Y 225.689,Z 778.242,A -85,B 0,C 180,E1 -19888.213,E2 -19888.213} C_VEL
LIN {X 0,Y 225.757,Z 779.031,A -85,B 0,C 180,E1 -19889.997,E2 -19889.997} C_VEL
LIN {X 0,Y 225.658,Z 779.38,A -85,B 0,C 180,E1 -19891.782,E2 -19891.782} C_VEL
LIN {X 0,Y 225.648,Z 778.9,A -85,B 0,C 180,E1 -19895.359,E2 -19895.359} C_VEL
LIN {X 0,Y 225.825,Z 778.056,A -85,B 0,C 180,E1 -19897.148,E2 -19897.148} C_VEL
LIN {X 0,Y 226.653,Z 775.098,A -85,B 0,C 180,E1 -19900.719,E2 -19900.719} C_VEL
LIN {X 0,Y 227.716,Z 771.757,A -85,B 0,C 180,E1 -19903.381,E2 -19903.381} C_VEL
LIN {X 0,Y 229.322,Z 767.374,A -85,B 0,C 180,E1 -19906.008,E2 -19906.008} C_VEL
LIN {X 0,Y 231.823,Z 760.794,A -85,B 0,C 180,E1 -19909.017,E2 -19909.017} C_VEL
LIN {X 0,Y 234.059,Z 754.055,A -85,B 0,C 180,E1 -19911.434,E2 -19911.434} C_VEL
LIN {X 0,Y 236.725,Z 746.377,A -85,B 0,C 180,E1 -19913.625,E2 -19913.625} C_VEL
LIN {X 0,Y 239.564,Z 737.635,A -85,B 0,C 180,E1 -19915.637,E2 -19915.637} C_VEL
LIN {X 0,Y 242.692,Z 726.957,A -85,B 0,C 180,E1 -19917.6,E2 -19917.6} C_VEL
LIN {X 0,Y 245.474,Z 716.431,A -85,B 0,C 180,E1 -19919.122,E2 -19919.122} C_VEL
LIN {X 0,Y 248.037,Z 704.808,A -85,B 0,C 180,E1 -19920.427,E2 -19920.427} C_VEL
LIN {X 0,Y 250.422,Z 691.719,A -85,B 0,C 180,E1 -19921.511,E2 -19921.511} C_VEL
LIN {X 0,Y 252.092,Z 679.462,A -85,B 0,C 180,E1 -19922.221,E2 -19922.221} C_VEL
LIN {X 0,Y 253.22,Z 664.563,A -85,B 0,C 180,E1 -19922.776,E2 -19922.776} C_VEL
LIN {X 0,Y 255.734,Z 621.876,A -85,B 0,C 180,E1 -19924.11,E2 -19924.11} C_VEL
LIN {X 0,Y 254.131,Z 609.113,A -85,B 0,C 180,E1 -19924.996,E2 -19924.996} C_VEL
LIN {X 0,Y 250.234,Z 599.741,A -85,B 0,C 180,E1 -19926.288,E2 -19926.288} C_VEL
LIN {X 0,Y 244.901,Z 588.942,A -85,B 0,C 180,E1 -19928.085,E2 -19928.085} C_VEL
LIN {X 0,Y 240.348,Z 580.668,A -85,B 0,C 180,E1 -19929.732,E2 -19929.732} C_VEL
LIN {X 0,Y 237.472,Z 575.837,A -85,B 0,C 180,E1 -19930.817,E2 -19930.817} C_VEL
LIN {X 0,Y 234.027,Z 570.452,A -85,B 0,C 180,E1 -19932.201,E2 -19932.201} C_VEL
LIN {X 0,Y 231.229,Z 566.471,A -85,B 0,C 180,E1 -19933.378,E2 -19933.378} C_VEL
LIN {X 0,Y 230.59,Z 565.116,A -85,B 0,C 180,E1 -19933.724,E2 -19933.724} C_VEL
LIN {X 0,Y 229.064,Z 560.071,A -85,B 0,C 180,E1 -19937.545,E2 -19937.545} C_VEL
LIN {X 0,Y 227.911,Z 556.097,A -85,B 0,C 180,E1 -19941.163,E2 -19941.163} C_VEL
LIN {X 0,Y 227.895,Z 556.099,A -85,B 0,C 180,E1 -19944.13,E2 -19944.13} C_VEL
LIN {X 0,Y 227.865,Z 556.095,A -85,B 0,C 180,E1 -19948.376,E2 -19948.376} C_VEL
LIN {X 0,Y 227.878,Z 556.09,A -85,B 0,C 180,E1 -19952.443,E2 -19952.443} C_VEL
LIN {X 0,Y 227.906,Z 556.085,A -85,B 0,C 180,E1 -19956.366,E2 -19956.366} C_VEL
LIN {X 0,Y 227.933,Z 556.081,A -85,B 0,C 180,E1 -19960.173,E2 -19960.173} C_VEL
LIN {X 0,Y 228.048,Z 556.067,A -85,B 0,C 180,E1 -19963.896,E2 -19963.896} C_VEL
LIN {X 0,Y 228.162,Z 556.059,A -85,B 0,C 180,E1 -19969.349,E2 -19969.349} C_VEL
LIN {X 0,Y 228.348,Z 556.036,A -85,B 0,C 180,E1 -19972.927,E2 -19972.927} C_VEL
LIN {X 0,Y 228.547,Z 556.009,A -85,B 0,C 180,E1 -19978.237,E2 -19978.237} C_VEL
LIN {X 0,Y 228.553,Z 556.009,A -85,B 0,C 180,E1 -19981.761,E2 -19981.761} C_VEL
LIN {X 0,Y 228.276,Z 556.088,A -85,B 0,C 180,E1 -19983.529,E2 -19983.529} C_VEL
LIN {X 0,Y 229.156,Z 558.806,A -85,B 0,C 180,E1 -19985.885,E2 -19985.885} C_VEL
LIN {X 0,Y 231.659,Z 562.544,A -85,B 0,C 180,E1 -19987.022,E2 -19987.022} C_VEL
LIN {X 0,Y 233.324,Z 564.553,A -85,B 0,C 180,E1 -19987.711,E2 -19987.711} C_VEL
LIN {X 0,Y 237.263,Z 570.647,A -85,B 0,C 180,E1 -19989.322,E2 -19989.322} C_VEL
LIN {X 0,Y 240.495,Z 575.59,A -85,B 0,C 180,E1 -19990.533,E2 -19990.533} C_VEL
LIN {X 0,Y 245.213,Z 583.364,A -85,B 0,C 180,E1 -19992.206,E2 -19992.206} C_VEL
LIN {X 0,Y 250.531,Z 593.341,A -85,B 0,C 180,E1 -19993.972,E2 -19993.972} C_VEL
LIN {X 0,Y 255.607,Z 604.654,A -85,B 0,C 180,E1 -19995.609,E2 -19995.609} C_VEL
LIN {X 0,Y 256.49,Z 607.251,A -85,B 0,C 180,E1 -19995.902,E2 -19995.902} C_VEL
LIN {X 0,Y 252.976,Z 664.331,A -85,B 0,C 180,E1 -19997.712,E2 -19997.712} C_VEL
LIN {X 0,Y 251.52,Z 677.323,A -85,B 0,C 180,E1 -19998.394,E2 -19998.394} C_VEL
LIN {X 0,Y 249.585,Z 690.089,A -85,B 0,C 180,E1 -19999.386,E2 -19999.386} C_VEL
LIN {X 0,Y 247.16,Z 702.254,A -85,B 0,C 180,E1 -20000.682,E2 -20000.682} C_VEL
LIN {X 0,Y 244.372,Z 713.778,A -85,B 0,C 180,E1 -20002.285,E2 -20002.285} C_VEL
LIN {X 0,Y 241.659,Z 723.603,A -85,B 0,C 180,E1 -20004.025,E2 -20004.025} C_VEL
LIN {X 0,Y 239.004,Z 732.04,A -85,B 0,C 180,E1 -20005.864,E2 -20005.864} C_VEL
LIN {X 0,Y 236.112,Z 740.419,A -85,B 0,C 180,E1 -20008.142,E2 -20008.142} C_VEL
LIN {X 0,Y 233.286,Z 748.13,A -85,B 0,C 180,E1 -20010.806,E2 -20010.806} C_VEL
LIN {X 0,Y 231.167,Z 753.535,A -85,B 0,C 180,E1 -20013.177,E2 -20013.177} C_VEL
LIN {X 0,Y 229.405,Z 757.897,A -85,B 0,C 180,E1 -20015.596,E2 -20015.596} C_VEL
LIN {X 0,Y 228.036,Z 761.31,A -85,B 0,C 180,E1 -20018.052,E2 -20018.052} C_VEL
LIN {X 0,Y 226.996,Z 763.874,A -85,B 0,C 180,E1 -20020.554,E2 -20020.554} C_VEL
LIN {X 0,Y 226.184,Z 765.634,A -85,B 0,C 180,E1 -20023.123,E2 -20023.123} C_VEL
LIN {X 0,Y 225.458,Z 766.627,A -85,B 0,C 180,E1 -20026.706,E2 -20026.706} C_VEL
LIN {X 0,Y 225.273,Z 766.423,A -85,B 0,C 180,E1 -20029.073,E2 -20029.073} C_VEL
LIN {X 0,Y 225.242,Z 765.526,A -85,B 0,C 180,E1 -20031.392,E2 -20031.392} C_VEL
LIN {X 0,Y 225.477,Z 763.564,A -85,B 0,C 180,E1 -20034.134,E2 -20034.134} C_VEL
LIN {X 0,Y 226.026,Z 760.316,A -85,B 0,C 180,E1 -20037.089,E2 -20037.089} C_VEL
LIN {X 0,Y 226.843,Z 755.282,A -85,B 0,C 180,E1 -20040.287,E2 -20040.287} C_VEL
LIN {X 0,Y 228.029,Z 748.81,A -85,B 0,C 180,E1 -20043.352,E2 -20043.352} C_VEL
LIN {X 0,Y 229.503,Z 741.404,A -85,B 0,C 180,E1 -20046.066,E2 -20046.066} C_VEL
LIN {X 0,Y 231.3,Z 732.567,A -85,B 0,C 180,E1 -20048.619,E2 -20048.619} C_VEL
LIN {X 0,Y 233.173,Z 722.84,A -85,B 0,C 180,E1 -20050.869,E2 -20050.869} C_VEL
LIN {X 0,Y 235.132,Z 712.039,A -85,B 0,C 180,E1 -20052.836,E2 -20052.836} C_VEL
LIN {X 0,Y 236.951,Z 700.346,A -85,B 0,C 180,E1 -20054.52,E2 -20054.52} C_VEL
LIN {X 0,Y 238.539,Z 688.658,A -85,B 0,C 180,E1 -20055.813,E2 -20055.813} C_VEL
LIN {X 0,Y 239.843,Z 675.632,A -85,B 0,C 180,E1 -20056.877,E2 -20056.877} C_VEL
LIN {X 0,Y 240.884,Z 662.355,A -85,B 0,C 180,E1 -20057.604,E2 -20057.604} C_VEL
LIN {X 0,Y 243.582,Z 596.06,A -85,B 0,C 180,E1 -20059.752,E2 -20059.752} C_VEL
LIN {X 0,Y 236.573,Z 576.588,A -85,B 0,C 180,E1 -20061.228,E2 -20061.228} C_VEL
LIN {X 0,Y 229.636,Z 559.326,A -85,B 0,C 180,E1 -20062.719,E2 -20062.719} C_VEL
LIN {X 0,Y 228.408,Z 556.408,A -85,B 0,C 180,E1 -20062.988,E2 -20062.988} C_VEL
LIN {X 0,Y 228.361,Z 556.042,A -85,B 0,C 180,E1 -20063.042,E2 -20063.042} C_VEL
LIN {X 0,Y 228.552,Z 556.015,A -85,B 0,C 180,E1 -20068.24,E2 -20068.24} C_VEL
LIN {X 0,Y 228.552,Z 556.013,A -85,B 0,C 180,E1 -20071.765,E2 -20071.765} C_VEL
LIN {X 0,Y 228.352,Z 556.038,A -85,B 0,C 180,E1 -20077.074,E2 -20077.074} C_VEL
LIN {X 0,Y 228.162,Z 556.063,A -85,B 0,C 180,E1 -20080.653,E2 -20080.653} C_VEL
LIN {X 0,Y 228.064,Z 556.069,A -85,B 0,C 180,E1 -20084.275,E2 -20084.275} C_VEL
LIN {X 0,Y 228.003,Z 556.082,A -85,B 0,C 180,E1 -20087.956,E2 -20087.956} C_VEL
LIN {X 0,Y 227.931,Z 556.072,A -85,B 0,C 180,E1 -20092.332,E2 -20092.332} C_VEL
LIN {X 0,Y 227.943,Z 556.088,A -85,B 0,C 180,E1 -20096.605,E2 -20096.605} C_VEL
LIN {X 0,Y 227.898,Z 556.095,A -85,B 0,C 180,E1 -20100.293,E2 -20100.293} C_VEL
LIN {X 0,Y 227.879,Z 556.098,A -85,B 0,C 180,E1 -20103.723,E2 -20103.723} C_VEL
LIN {X 0,Y 227.846,Z 556.101,A -85,B 0,C 180,E1 -20108.093,E2 -20108.093} C_VEL
LIN {X 0,Y 227.816,Z 556.102,A -85,B 0,C 180,E1 -20112.744,E2 -20112.744} C_VEL
LIN {X 0,Y 227.817,Z 556.107,A -85,B 0,C 180,E1 -20117.26,E2 -20117.26} C_VEL
LIN {X 0,Y 227.848,Z 556.098,A -85,B 0,C 180,E1 -20121.911,E2 -20121.911} C_VEL
LIN {X 0,Y 227.885,Z 556.097,A -85,B 0,C 180,E1 -20126.379,E2 -20126.379} C_VEL
LIN {X 0,Y 227.925,Z 556.082,A -85,B 0,C 180,E1 -20130.44,E2 -20130.44} C_VEL
LIN {X 0,Y 227.931,Z 556.088,A -85,B 0,C 180,E1 -20134.427,E2 -20134.427} C_VEL
LIN {X 0,Y 227.951,Z 556.087,A -85,B 0,C 180,E1 -20138.287,E2 -20138.287} C_VEL
LIN {X 0,Y 228.015,Z 556.067,A -85,B 0,C 180,E1 -20142.849,E2 -20142.849} C_VEL
LIN {X 0,Y 228.075,Z 556.075,A -85,B 0,C 180,E1 -20147.544,E2 -20147.544} C_VEL
LIN {X 0,Y 228.276,Z 556.046,A -85,B 0,C 180,E1 -20151.146,E2 -20151.146} C_VEL
LIN {X 0,Y 228.332,Z 556.032,A -85,B 0,C 180,E1 -20152.929,E2 -20152.929} C_VEL
LIN {X 0,Y 228.562,Z 556.014,A -85,B 0,C 180,E1 -20158.239,E2 -20158.239} C_VEL
LIN {X 0,Y 228.563,Z 556.011,A -85,B 0,C 180,E1 -20161.763,E2 -20161.763} C_VEL
LIN {X 0,Y 228.367,Z 556.036,A -85,B 0,C 180,E1 -20167.072,E2 -20167.072} C_VEL
LIN {X 0,Y 228.177,Z 556.059,A -85,B 0,C 180,E1 -20170.651,E2 -20170.651} C_VEL
LIN {X 0,Y 228.074,Z 556.073,A -85,B 0,C 180,E1 -20174.272,E2 -20174.272} C_VEL
LIN {X 0,Y 228.012,Z 556.085,A -85,B 0,C 180,E1 -20177.953,E2 -20177.953} C_VEL
LIN {X 0,Y 227.926,Z 556.076,A -85,B 0,C 180,E1 -20182.321,E2 -20182.321} C_VEL
LIN {X 0,Y 227.945,Z 556.083,A -85,B 0,C 180,E1 -20186.666,E2 -20186.666} C_VEL
LIN {X 0,Y 227.906,Z 556.096,A -85,B 0,C 180,E1 -20190.291,E2 -20190.291} C_VEL
LIN {X 0,Y 227.858,Z 556.098,A -85,B 0,C 180,E1 -20194.353,E2 -20194.353} C_VEL
LIN {X 0,Y 227.168,Z 556.189,A -85,B 0,C 180,E1 -20195.829,E2 -20195.829} C_VEL
LIN {X 0,Y 224.316,Z 556.546,A -85,B 0,C 180,E1 -20198.238,E2 -20198.238} C_VEL
LIN {X 0,Y 221.901,Z 556.848,A -85,B 0,C 180,E1 -20200.204,E2 -20200.204} C_VEL
LIN {X 0,Y 220.859,Z 556.975,A -85,B 0,C 180,E1 -20201.729,E2 -20201.729} C_VEL
LIN {X 0,Y 220.77,Z 556.984,A -85,B 0,C 180,E1 -20202.246,E2 -20202.246} C_VEL
LIN {X 0,Y 220.779,Z 556.978,A -85,B 0,C 180,E1 -20205.544,E2 -20205.544} C_VEL
LIN {X 0,Y 220.818,Z 556.981,A -85,B 0,C 180,E1 -20210.463,E2 -20210.463} C_VEL
LIN {X 0,Y 220.902,Z 557.104,A -85,B 0,C 180,E1 -20211.616,E2 -20211.616} C_VEL
LIN {X 0,Y 222.723,Z 565.346,A -85,B 0,C 180,E1 -20215.387,E2 -20215.387} C_VEL
LIN {X 0,Y 223.207,Z 567.623,A -85,B 0,C 180,E1 -20216.348,E2 -20216.348} C_VEL
LIN {X 0,Y 232.786,Z 592.85,A -85,B 0,C 180,E1 -20218.507,E2 -20218.507} C_VEL
LIN {X 0,Y 234.186,Z 601.748,A -85,B 0,C 180,E1 -20219.004,E2 -20219.004} C_VEL
LIN {X 0,Y 236.474,Z 620.167,A -85,B 0,C 180,E1 -20219.943,E2 -20219.943} C_VEL
LIN {X 0,Y 234.028,Z 676.351,A -85,B 0,C 180,E1 -20221.83,E2 -20221.83} C_VEL
LIN {X 0,Y 232.834,Z 689.631,A -85,B 0,C 180,E1 -20222.59,E2 -20222.59} C_VEL
LIN {X 0,Y 231.307,Z 701.913,A -85,B 0,C 180,E1 -20223.615,E2 -20223.615} C_VEL
LIN {X 0,Y 229.686,Z 713.048,A -85,B 0,C 180,E1 -20224.875,E2 -20224.875} C_VEL
LIN {X 0,Y 227.763,Z 724.698,A -85,B 0,C 180,E1 -20226.589,E2 -20226.589} C_VEL
LIN {X 0,Y 225.913,Z 734.113,A -85,B 0,C 180,E1 -20228.317,E2 -20228.317} C_VEL
LIN {X 0,Y 224.022,Z 743.4,A -85,B 0,C 180,E1 -20230.423,E2 -20230.423} C_VEL
LIN {X 0,Y 222.547,Z 750.982,A -85,B 0,C 180,E1 -20232.539,E2 -20232.539} C_VEL
LIN {X 0,Y 220.965,Z 758.859,A -85,B 0,C 180,E1 -20235.257,E2 -20235.257} C_VEL
LIN {X 0,Y 219.789,Z 765.146,A -85,B 0,C 180,E1 -20238.001,E2 -20238.001} C_VEL
LIN {X 0,Y 219.085,Z 770.118,A -85,B 0,C 180,E1 -20240.768,E2 -20240.768} C_VEL
LIN {X 0,Y 218.703,Z 773.913,A -85,B 0,C 180,E1 -20243.54,E2 -20243.54} C_VEL
LIN {X 0,Y 218.528,Z 776.636,A -85,B 0,C 180,E1 -20246.31,E2 -20246.31} C_VEL
LIN {X 0,Y 218.604,Z 777.906,A -85,B 0,C 180,E1 -20248.155,E2 -20248.155} C_VEL
LIN {X 0,Y 218.669,Z 778.76,A -85,B 0,C 180,E1 -20249.997,E2 -20249.997} C_VEL
LIN {X 0,Y 218.555,Z 779.153,A -85,B 0,C 180,E1 -20251.84,E2 -20251.84} C_VEL
LIN {X 0,Y 218.515,Z 779.059,A -85,B 0,C 180,E1 -20254.4,E2 -20254.4} C_VEL
LIN {X 0,Y 218.763,Z 777.957,A -85,B 0,C 180,E1 -20257.38,E2 -20257.38} C_VEL
LIN {X 0,Y 219.109,Z 776.736,A -85,B 0,C 180,E1 -20259.226,E2 -20259.226} C_VEL
LIN {X 0,Y 219.991,Z 774.151,A -85,B 0,C 180,E1 -20261.982,E2 -20261.982} C_VEL
LIN {X 0,Y 221.252,Z 770.569,A -85,B 0,C 180,E1 -20264.718,E2 -20264.718} C_VEL
LIN {X 0,Y 223.221,Z 765.899,A -85,B 0,C 180,E1 -20267.401,E2 -20267.401} C_VEL
LIN {X 0,Y 225.919,Z 758.885,A -85,B 0,C 180,E1 -20270.483,E2 -20270.483} C_VEL
LIN {X 0,Y 228.632,Z 751.356,A -85,B 0,C 180,E1 -20273.071,E2 -20273.071} C_VEL
LIN {X 0,Y 231.413,Z 743.73,A -85,B 0,C 180,E1 -20275.159,E2 -20275.159} C_VEL
LIN {X 0,Y 234.56,Z 734.532,A -85,B 0,C 180,E1 -20277.186,E2 -20277.186} C_VEL
LIN {X 0,Y 237.487,Z 724.408,A -85,B 0,C 180,E1 -20278.982,E2 -20278.982} C_VEL
LIN {X 0,Y 240.507,Z 713.255,A -85,B 0,C 180,E1 -20280.509,E2 -20280.509} C_VEL
LIN {X 0,Y 243.232,Z 700.87,A -85,B 0,C 180,E1 -20281.821,E2 -20281.821} C_VEL
LIN {X 0,Y 245.52,Z 687.614,A -85,B 0,C 180,E1 -20282.823,E2 -20282.823} C_VEL
LIN {X 0,Y 247.217,Z 674.449,A -85,B 0,C 180,E1 -20283.481,E2 -20283.481} C_VEL
LIN {X 0,Y 250.42,Z 622.864,A -85,B 0,C 180,E1 -20285.175,E2 -20285.175} C_VEL
LIN {X 0,Y 249.207,Z 612.284,A -85,B 0,C 180,E1 -20285.933,E2 -20285.933} C_VEL
LIN {X 0,Y 245.297,Z 602.787,A -85,B 0,C 180,E1 -20287.302,E2 -20287.302} C_VEL
LIN {X 0,Y 239.513,Z 590.872,A -85,B 0,C 180,E1 -20289.422,E2 -20289.422} C_VEL
LIN {X 0,Y 234.273,Z 581.588,A -85,B 0,C 180,E1 -20291.47,E2 -20291.47} C_VEL
LIN {X 0,Y 230.737,Z 576.023,A -85,B 0,C 180,E1 -20292.956,E2 -20292.956} C_VEL
LIN {X 0,Y 227.738,Z 571.415,A -85,B 0,C 180,E1 -20294.309,E2 -20294.309} C_VEL
LIN {X 0,Y 223.891,Z 566.074,A -85,B 0,C 180,E1 -20296.183,E2 -20296.183} C_VEL
LIN {X 0,Y 223.268,Z 564.684,A -85,B 0,C 180,E1 -20296.589,E2 -20296.589} C_VEL
LIN {X 0,Y 221.782,Z 560.088,A -85,B 0,C 180,E1 -20300.67,E2 -20300.67} C_VEL
LIN {X 0,Y 220.847,Z 556.974,A -85,B 0,C 180,E1 -20303.932,E2 -20303.932} C_VEL
LIN {X 0,Y 220.856,Z 556.965,A -85,B 0,C 180,E1 -20309.219,E2 -20309.219} C_VEL
LIN {X 0,Y 220.887,Z 556.962,A -85,B 0,C 180,E1 -20313.548,E2 -20313.548} C_VEL
LIN {X 0,Y 220.869,Z 556.965,A -85,B 0,C 180,E1 -20317.552,E2 -20317.552} C_VEL
LIN {X 0,Y 220.975,Z 556.96,A -85,B 0,C 180,E1 -20322.569,E2 -20322.569} C_VEL
LIN {X 0,Y 221.017,Z 556.947,A -85,B 0,C 180,E1 -20327.138,E2 -20327.138} C_VEL
LIN {X 0,Y 221.248,Z 556.919,A -85,B 0,C 180,E1 -20330.86,E2 -20330.86} C_VEL
LIN {X 0,Y 221.285,Z 556.913,A -85,B 0,C 180,E1 -20332.701,E2 -20332.701} C_VEL
LIN {X 0,Y 221.505,Z 556.887,A -85,B 0,C 180,E1 -20338.181,E2 -20338.181} C_VEL
LIN {X 0,Y 221.535,Z 557.012,A -85,B 0,C 180,E1 -20340.908,E2 -20340.908} C_VEL
LIN {X 0,Y 222.004,Z 559.217,A -85,B 0,C 180,E1 -20343.005,E2 -20343.005} C_VEL
LIN {X 0,Y 224.775,Z 563.332,A -85,B 0,C 180,E1 -20344.483,E2 -20344.483} C_VEL
LIN {X 0,Y 226.474,Z 565.164,A -85,B 0,C 180,E1 -20345.286,E2 -20345.286} C_VEL
LIN {X 0,Y 229.532,Z 569.312,A -85,B 0,C 180,E1 -20346.703,E2 -20346.703} C_VEL
LIN {X 0,Y 233.779,Z 575.932,A -85,B 0,C 180,E1 -20348.535,E2 -20348.535} C_VEL
LIN {X 0,Y 237.515,Z 581.855,A -85,B 0,C 180,E1 -20350.024,E2 -20350.024} C_VEL
LIN {X 0,Y 242.808,Z 590.991,A -85,B 0,C 180,E1 -20351.969,E2 -20351.969} C_VEL
LIN {X 0,Y 247.952,Z 601.488,A -85,B 0,C 180,E1 -20353.761,E2 -20353.761} C_VEL
LIN {X 0,Y 251.223,Z 609.228,A -85,B 0,C 180,E1 -20354.868,E2 -20354.868} C_VEL
LIN {X 0,Y 247.511,Z 665.128,A -85,B 0,C 180,E1 -20356.681,E2 -20356.681} C_VEL
LIN {X 0,Y 245.945,Z 678.409,A -85,B 0,C 180,E1 -20357.406,E2 -20357.406} C_VEL
LIN {X 0,Y 244.009,Z 690.546,A -85,B 0,C 180,E1 -20358.377,E2 -20358.377} C_VEL
LIN {X 0,Y 241.315,Z 703.255,A -85,B 0,C 180,E1 -20359.763,E2 -20359.763} C_VEL
LIN {X 0,Y 238.443,Z 714.601,A -85,B 0,C 180,E1 -20361.391,E2 -20361.391} C_VEL
LIN {X 0,Y 235.355,Z 724.998,A -85,B 0,C 180,E1 -20363.306,E2 -20363.306} C_VEL
LIN {X 0,Y 232.064,Z 734.67,A -85,B 0,C 180,E1 -20365.564,E2 -20365.564} C_VEL
LIN {X 0,Y 229.117,Z 742.565,A -85,B 0,C 180,E1 -20367.888,E2 -20367.888} C_VEL
LIN {X 0,Y 226.543,Z 749.132,A -85,B 0,C 180,E1 -20370.319,E2 -20370.319} C_VEL
LIN {X 0,Y 223.847,Z 755.536,A -85,B 0,C 180,E1 -20373.383,E2 -20373.383} C_VEL
LIN {X 0,Y 222.086,Z 759.566,A -85,B 0,C 180,E1 -20375.907,E2 -20375.907} C_VEL
LIN {X 0,Y 220.671,Z 762.802,A -85,B 0,C 180,E1 -20378.612,E2 -20378.612} C_VEL
LIN {X 0,Y 220.11,Z 764.058,A -85,B 0,C 180,E1 -20379.981,E2 -20379.981} C_VEL
LIN {X 0,Y 219.251,Z 765.758,A -85,B 0,C 180,E1 -20382.506,E2 -20382.506} C_VEL
LIN {X 0,Y 218.649,Z 766.651,A -85,B 0,C 180,E1 -20385.001,E2 -20385.001} C_VEL
LIN {X 0,Y 218.237,Z 766.803,A -85,B 0,C 180,E1 -20387.788,E2 -20387.788} C_VEL
LIN {X 0,Y 218.151,Z 766.01,A -85,B 0,C 180,E1 -20390.639,E2 -20390.639} C_VEL
LIN {X 0,Y 218.303,Z 764.156,A -85,B 0,C 180,E1 -20393.593,E2 -20393.593} C_VEL
LIN {X 0,Y 218.869,Z 760.753,A -85,B 0,C 180,E1 -20396.919,E2 -20396.919} C_VEL
LIN {X 0,Y 219.58,Z 756.579,A -85,B 0,C 180,E1 -20399.787,E2 -20399.787} C_VEL
LIN {X 0,Y 220.482,Z 751.857,A -85,B 0,C 180,E1 -20402.288,E2 -20402.288} C_VEL
LIN {X 0,Y 221.851,Z 744.955,A -85,B 0,C 180,E1 -20405.185,E2 -20405.185} C_VEL
LIN {X 0,Y 223.483,Z 736.932,A -85,B 0,C 180,E1 -20407.832,E2 -20407.832} C_VEL
LIN {X 0,Y 225.315,Z 728.087,A -85,B 0,C 180,E1 -20410.174,E2 -20410.174} C_VEL
LIN {X 0,Y 227.177,Z 718.444,A -85,B 0,C 180,E1 -20412.234,E2 -20412.234} C_VEL
LIN {X 0,Y 229.287,Z 706.603,A -85,B 0,C 180,E1 -20414.218,E2 -20414.218} C_VEL
LIN {X 0,Y 231.079,Z 694.413,A -85,B 0,C 180,E1 -20415.808,E2 -20415.808} C_VEL
LIN {X 0,Y 232.665,Z 681.817,A -85,B 0,C 180,E1 -20417.02,E2 -20417.02} C_VEL
LIN {X 0,Y 233.836,Z 668.786,A -85,B 0,C 180,E1 -20417.918,E2 -20417.918} C_VEL
LIN {X 0,Y 234.674,Z 654.878,A -85,B 0,C 180,E1 -20418.504,E2 -20418.504} C_VEL
LIN {X 0,Y 236.994,Z 597.51,A -85,B 0,C 180,E1 -20420.394,E2 -20420.394} C_VEL
LIN {X 0,Y 230.454,Z 579.194,A -85,B 0,C 180,E1 -20421.84,E2 -20421.84} C_VEL
LIN {X 0,Y 223.986,Z 563.097,A -85,B 0,C 180,E1 -20423.274,E2 -20423.274} C_VEL
LIN {X 0,Y 221.39,Z 557.807,A -85,B 0,C 180,E1 -20423.824,E2 -20423.824} C_VEL
LIN {X 0,Y 221.199,Z 556.936,A -85,B 0,C 180,E1 -20423.961,E2 -20423.961} C_VEL
LIN {X 0,Y 221.51,Z 556.892,A -85,B 0,C 180,E1 -20428.184,E2 -20428.184} C_VEL
LIN {X 0,Y 221.51,Z 556.891,A -85,B 0,C 180,E1 -20431.821,E2 -20431.821} C_VEL
LIN {X 0,Y 221.303,Z 556.918,A -85,B 0,C 180,E1 -20437.301,E2 -20437.301} C_VEL
LIN {X 0,Y 221.111,Z 556.937,A -85,B 0,C 180,E1 -20440.997,E2 -20440.997} C_VEL
LIN {X 0,Y 221.017,Z 556.954,A -85,B 0,C 180,E1 -20446.632,E2 -20446.632} C_VEL
LIN {X 0,Y 220.893,Z 556.959,A -85,B 0,C 180,E1 -20450.489,E2 -20450.489} C_VEL
LIN {X 0,Y 220.868,Z 556.961,A -85,B 0,C 180,E1 -20454.437,E2 -20454.437} C_VEL
LIN {X 0,Y 220.829,Z 556.978,A -85,B 0,C 180,E1 -20458.517,E2 -20458.517} C_VEL
LIN {X 0,Y 220.818,Z 556.972,A -85,B 0,C 180,E1 -20462.759,E2 -20462.759} C_VEL
LIN {X 0,Y 220.813,Z 556.981,A -85,B 0,C 180,E1 -20467.281,E2 -20467.281} C_VEL
LIN {X 0,Y 220.774,Z 556.979,A -85,B 0,C 180,E1 -20471.955,E2 -20471.955} C_VEL
LIN {X 0,Y 220.779,Z 556.985,A -85,B 0,C 180,E1 -20475.549,E2 -20475.549} C_VEL
LIN {X 0,Y 220.811,Z 556.966,A -85,B 0,C 180,E1 -20480.465,E2 -20480.465} C_VEL
LIN {X 0,Y 220.806,Z 556.979,A -85,B 0,C 180,E1 -20485.047,E2 -20485.047} C_VEL
LIN {X 0,Y 220.874,Z 556.965,A -85,B 0,C 180,E1 -20489.397,E2 -20489.397} C_VEL
LIN {X 0,Y 220.901,Z 556.962,A -85,B 0,C 180,E1 -20493.551,E2 -20493.551} C_VEL
LIN {X 0,Y 220.871,Z 556.974,A -85,B 0,C 180,E1 -20497.554,E2 -20497.554} C_VEL
LIN {X 0,Y 220.969,Z 556.944,A -85,B 0,C 180,E1 -20502.591,E2 -20502.591} C_VEL
LIN {X 0,Y 221.012,Z 556.952,A -85,B 0,C 180,E1 -20507.14,E2 -20507.14} C_VEL
LIN {X 0,Y 221.213,Z 556.925,A -85,B 0,C 180,E1 -20510.861,E2 -20510.861} C_VEL
LIN {X 0,Y 221.268,Z 556.911,A -85,B 0,C 180,E1 -20512.702,E2 -20512.702} C_VEL
LIN {X 0,Y 221.52,Z 556.891,A -85,B 0,C 180,E1 -20518.183,E2 -20518.183} C_VEL
LIN {X 0,Y 221.521,Z 556.887,A -85,B 0,C 180,E1 -20521.819,E2 -20521.819} C_VEL
LIN {X 0,Y 221.32,Z 556.914,A -85,B 0,C 180,E1 -20527.298,E2 -20527.298} C_VEL
LIN {X 0,Y 221.121,Z 556.937,A -85,B 0,C 180,E1 -20530.995,E2 -20530.995} C_VEL
LIN {X 0,Y 221.026,Z 556.953,A -85,B 0,C 180,E1 -20536.63,E2 -20536.63} C_VEL
LIN {X 0,Y 220.894,Z 556.961,A -85,B 0,C 180,E1 -20540.487,E2 -20540.487} C_VEL
LIN {X 0,Y 220.872,Z 556.949,A -85,B 0,C 180,E1 -20544.435,E2 -20544.435} C_VEL
LIN {X 0,Y 220.836,Z 556.976,A -85,B 0,C 180,E1 -20548.515,E2 -20548.515} C_VEL
LIN {X 0,Y 220.828,Z 556.977,A -85,B 0,C 180,E1 -20552.755,E2 -20552.755} C_VEL
LIN {X 0,Y 220.82,Z 556.978,A -85,B 0,C 180,E1 -20557.278,E2 -20557.278} C_VEL
LIN {X 0,Y 220.778,Z 556.984,A -85,B 0,C 180,E1 -20561.952,E2 -20561.952} C_VEL
LIN {X 0,Y 220.77,Z 556.984,A -85,B 0,C 180,E1 -20562.246,E2 -20562.246} C_VEL
LIN {X 0,Y 220.087,Z 557.07,A -85,B 0,C 180,E1 -20563.767,E2 -20563.767} C_VEL
LIN {X 0,Y 217.229,Z 557.425,A -85,B 0,C 180,E1 -20566.249,E2 -20566.249} C_VEL
LIN {X 0,Y 214.834,Z 557.724,A -85,B 0,C 180,E1 -20568.276,E2 -20568.276} C_VEL
LIN {X 0,Y 213.845,Z 557.847,A -85,B 0,C 180,E1 -20569.85,E2 -20569.85} C_VEL
LIN {X 0,Y 213.785,Z 557.855,A -85,B 0,C 180,E1 -20570.383,E2 -20570.383} C_VEL
LIN {X 0,Y 213.837,Z 558.001,A -85,B 0,C 180,E1 -20570.977,E2 -20570.977} C_VEL
LIN {X 0,Y 215.708,Z 566.271,A -85,B 0,C 180,E1 -20574.901,E2 -20574.901} C_VEL
LIN {X 0,Y 215.945,Z 567.401,A -85,B 0,C 180,E1 -20575.379,E2 -20575.379} C_VEL
LIN {X 0,Y 226.034,Z 593.582,A -85,B 0,C 180,E1 -20577.743,E2 -20577.743} C_VEL
LIN {X 0,Y 227.027,Z 597.136,A -85,B 0,C 180,E1 -20578.003,E2 -20578.003} C_VEL
LIN {X 0,Y 229.964,Z 620.757,A -85,B 0,C 180,E1 -20579.263,E2 -20579.263} C_VEL
LIN {X 0,Y 227.434,Z 676.437,A -85,B 0,C 180,E1 -20581.19,E2 -20581.19} C_VEL
LIN {X 0,Y 226.193,Z 689.609,A -85,B 0,C 180,E1 -20581.967,E2 -20581.967} C_VEL
LIN {X 0,Y 224.631,Z 701.844,A -85,B 0,C 180,E1 -20583.019,E2 -20583.019} C_VEL
LIN {X 0,Y 222.956,Z 712.942,A -85,B 0,C 180,E1 -20584.312,E2 -20584.312} C_VEL
LIN {X 0,Y 220.965,Z 724.575,A -85,B 0,C 180,E1 -20586.073,E2 -20586.073} C_VEL
LIN {X 0,Y 219.061,Z 733.979,A -85,B 0,C 180,E1 -20587.851,E2 -20587.851} C_VEL
LIN {X 0,Y 217.069,Z 743.382,A -85,B 0,C 180,E1 -20590.05,E2 -20590.05} C_VEL
LIN {X 0,Y 215.762,Z 750.078,A -85,B 0,C 180,E1 -20591.972,E2 -20591.972} C_VEL
LIN {X 0,Y 214.086,Z 758.126,A -85,B 0,C 180,E1 -20594.772,E2 -20594.772} C_VEL
LIN {X 0,Y 212.808,Z 764.515,A -85,B 0,C 180,E1 -20597.602,E2 -20597.602} C_VEL
LIN {X 0,Y 212.057,Z 769.581,A -85,B 0,C 180,E1 -20600.459,E2 -20600.459} C_VEL
LIN {X 0,Y 211.637,Z 773.461,A -85,B 0,C 180,E1 -20603.323,E2 -20603.323} C_VEL
LIN {X 0,Y 211.44,Z 776.263,A -85,B 0,C 180,E1 -20606.186,E2 -20606.186} C_VEL
LIN {X 0,Y 211.501,Z 777.57,A -85,B 0,C 180,E1 -20608.093,E2 -20608.093} C_VEL
LIN {X 0,Y 211.583,Z 778.463,A -85,B 0,C 180,E1 -20609.997,E2 -20609.997} C_VEL
LIN {X 0,Y 211.455,Z 778.925,A -85,B 0,C 180,E1 -20611.902,E2 -20611.902} C_VEL
LIN {X 0,Y 211.421,Z 778.906,A -85,B 0,C 180,E1 -20614.238,E2 -20614.238} C_VEL
LIN {X 0,Y 211.692,Z 777.849,A -85,B 0,C 180,E1 -20617.628,E2 -20617.628} C_VEL
LIN {X 0,Y 212.084,Z 776.705,A -85,B 0,C 180,E1 -20619.534,E2 -20619.534} C_VEL
LIN {X 0,Y 213.033,Z 774.187,A -85,B 0,C 180,E1 -20622.38,E2 -20622.38} C_VEL
LIN {X 0,Y 214.371,Z 770.678,A -85,B 0,C 180,E1 -20625.202,E2 -20625.202} C_VEL
LIN {X 0,Y 216.443,Z 766.106,A -85,B 0,C 180,E1 -20627.964,E2 -20627.964} C_VEL
LIN {X 0,Y 218.832,Z 760.372,A -85,B 0,C 180,E1 -20630.685,E2 -20630.685} C_VEL
LIN {X 0,Y 221.623,Z 753.241,A -85,B 0,C 180,E1 -20633.349,E2 -20633.349} C_VEL
LIN {X 0,Y 225.056,Z 744.398,A -85,B 0,C 180,E1 -20635.922,E2 -20635.922} C_VEL
LIN {X 0,Y 228.636,Z 734.406,A -85,B 0,C 180,E1 -20638.201,E2 -20638.201} C_VEL
LIN {X 0,Y 231.752,Z 724.291,A -85,B 0,C 180,E1 -20640.021,E2 -20640.021} C_VEL
LIN {X 0,Y 234.896,Z 713.189,A -85,B 0,C 180,E1 -20641.57,E2 -20641.57} C_VEL
LIN {X 0,Y 237.743,Z 700.926,A -85,B 0,C 180,E1 -20642.898,E2 -20642.898} C_VEL
LIN {X 0,Y 240.177,Z 687.463,A -85,B 0,C 180,E1 -20643.938,E2 -20643.938} C_VEL
LIN {X 0,Y 241.989,Z 673.935,A -85,B 0,C 180,E1 -20644.623,E2 -20644.623} C_VEL
LIN {X 0,Y 245.228,Z 623.503,A -85,B 0,C 180,E1 -20646.317,E2 -20646.317} C_VEL
LIN {X 0,Y 244.296,Z 615.161,A -85,B 0,C 180,E1 -20646.939,E2 -20646.939} C_VEL
LIN {X 0,Y 240.087,Z 605.144,A -85,B 0,C 180,E1 -20648.511,E2 -20648.511} C_VEL
LIN {X 0,Y 234.922,Z 594.439,A -85,B 0,C 180,E1 -20650.534,E2 -20650.534} C_VEL
LIN {X 0,Y 230.498,Z 586.46,A -85,B 0,C 180,E1 -20652.403,E2 -20652.403} C_VEL
LIN {X 0,Y 227.439,Z 581.491,A -85,B 0,C 180,E1 -20653.761,E2 -20653.761} C_VEL
LIN {X 0,Y 223.802,Z 575.884,A -85,B 0,C 180,E1 -20655.527,E2 -20655.527} C_VEL
LIN {X 0,Y 220.8,Z 571.336,A -85,B 0,C 180,E1 -20657.108,E2 -20657.108} C_VEL
LIN {X 0,Y 216.192,Z 565.062,A -85,B 0,C 180,E1 -20659.827,E2 -20659.827} C_VEL
LIN {X 0,Y 215.747,Z 564.1,A -85,B 0,C 180,E1 -20660.261,E2 -20660.261} C_VEL
LIN {X 0,Y 214.755,Z 560.651,A -85,B 0,C 180,E1 -20663.909,E2 -20663.909} C_VEL
LIN {X 0,Y 213.783,Z 557.855,A -85,B 0,C 180,E1 -20667.709,E2 -20667.709} C_VEL
LIN {X 0,Y 213.818,Z 557.84,A -85,B 0,C 180,E1 -20672.601,E2 -20672.601} C_VEL
LIN {X 0,Y 213.844,Z 557.837,A -85,B 0,C 180,E1 -20676.951,E2 -20676.951} C_VEL
LIN {X 0,Y 213.935,Z 557.833,A -85,B 0,C 180,E1 -20682.802,E2 -20682.802} C_VEL
LIN {X 0,Y 213.971,Z 557.829,A -85,B 0,C 180,E1 -20686.707,E2 -20686.707} C_VEL
LIN {X 0,Y 214.186,Z 557.802,A -85,B 0,C 180,E1 -20690.556,E2 -20690.556} C_VEL
LIN {X 0,Y 214.102,Z 557.811,A -85,B 0,C 180,E1 -20694.348,E2 -20694.348} C_VEL
LIN {X 0,Y 214.289,Z 557.871,A -85,B 0,C 180,E1 -20697.179,E2 -20697.179} C_VEL
LIN {X 0,Y 214.992,Z 559.596,A -85,B 0,C 180,E1 -20699.531,E2 -20699.531} C_VEL
LIN {X 0,Y 218.217,Z 564.048,A -85,B 0,C 180,E1 -20701.605,E2 -20701.605} C_VEL
LIN {X 0,Y 219.707,Z 565.823,A -85,B 0,C 180,E1 -20702.463,E2 -20702.463} C_VEL
LIN {X 0,Y 222.628,Z 569.973,A -85,B 0,C 180,E1 -20704.072,E2 -20704.072} C_VEL
LIN {X 0,Y 224.153,Z 571.899,A -85,B 0,C 180,E1 -20704.833,E2 -20704.833} C_VEL
LIN {X 0,Y 227.5,Z 576.621,A -85,B 0,C 180,E1 -20706.443,E2 -20706.443} C_VEL
LIN {X 0,Y 233.13,Z 585.676,A -85,B 0,C 180,E1 -20708.9,E2 -20708.9} C_VEL
LIN {X 0,Y 238.155,Z 594.553,A -85,B 0,C 180,E1 -20710.895,E2 -20710.895} C_VEL
LIN {X 0,Y 242.478,Z 603.317,A -85,B 0,C 180,E1 -20712.516,E2 -20712.516} C_VEL
LIN {X 0,Y 245.951,Z 611.423,A -85,B 0,C 180,E1 -20713.769,E2 -20713.769} C_VEL
LIN {X 0,Y 242.307,Z 665.248,A -85,B 0,C 180,E1 -20715.558,E2 -20715.558} C_VEL
LIN {X 0,Y 240.695,Z 678.351,A -85,B 0,C 180,E1 -20716.28,E2 -20716.28} C_VEL
LIN {X 0,Y 238.68,Z 690.298,A -85,B 0,C 180,E1 -20717.239,E2 -20717.239} C_VEL
LIN {X 0,Y 236.294,Z 701.302,A -85,B 0,C 180,E1 -20718.413,E2 -20718.413} C_VEL
LIN {X 0,Y 233.427,Z 712.218,A -85,B 0,C 180,E1 -20719.926,E2 -20719.926} C_VEL
LIN {X 0,Y 230.368,Z 722.559,A -85,B 0,C 180,E1 -20721.76,E2 -20721.76} C_VEL
LIN {X 0,Y 227.286,Z 731.423,A -85,B 0,C 180,E1 -20723.701,E2 -20723.701} C_VEL
LIN {X 0,Y 224.059,Z 739.951,A -85,B 0,C 180,E1 -20726.048,E2 -20726.048} C_VEL
LIN {X 0,Y 220.732,Z 747.951,A -85,B 0,C 180,E1 -20728.885,E2 -20728.885} C_VEL
LIN {X 0,Y 217.896,Z 754.348,A -85,B 0,C 180,E1 -20731.828,E2 -20731.828} C_VEL
LIN {X 0,Y 215.88,Z 758.642,A -85,B 0,C 180,E1 -20734.4,E2 -20734.4} C_VEL
LIN {X 0,Y 214.312,Z 761.98,A -85,B 0,C 180,E1 -20737.009,E2 -20737.009} C_VEL
LIN {X 0,Y 212.766,Z 765.133,A -85,B 0,C 180,E1 -20740.564,E2 -20740.564} C_VEL
LIN {X 0,Y 211.704,Z 766.777,A -85,B 0,C 180,E1 -20744.197,E2 -20744.197} C_VEL
LIN {X 0,Y 211.233,Z 767.063,A -85,B 0,C 180,E1 -20747.05,E2 -20747.05} C_VEL
LIN {X 0,Y 211.063,Z 766.075,A -85,B 0,C 180,E1 -20750.757,E2 -20750.757} C_VEL
LIN {X 0,Y 211.321,Z 763.614,A -85,B 0,C 180,E1 -20754.412,E2 -20754.412} C_VEL
LIN {X 0,Y 211.793,Z 760.821,A -85,B 0,C 180,E1 -20757.05,E2 -20757.05} C_VEL
LIN {X 0,Y 212.632,Z 756.142,A -85,B 0,C 180,E1 -20760.282,E2 -20760.282} C_VEL
LIN {X 0,Y 213.753,Z 750.479,A -85,B 0,C 180,E1 -20763.228,E2 -20763.228} C_VEL
LIN {X 0,Y 215.2,Z 743.394,A -85,B 0,C 180,E1 -20766.122,E2 -20766.122} C_VEL
LIN {X 0,Y 216.874,Z 735.726,A -85,B 0,C 180,E1 -20768.622,E2 -20768.622} C_VEL
LIN {X 0,Y 218.779,Z 726.576,A -85,B 0,C 180,E1 -20771.022,E2 -20771.022} C_VEL
LIN {X 0,Y 220.716,Z 716.961,A -85,B 0,C 180,E1 -20773.043,E2 -20773.043} C_VEL
LIN {X 0,Y 222.711,Z 705.855,A -85,B 0,C 180,E1 -20774.912,E2 -20774.912} C_VEL
LIN {X 0,Y 224.424,Z 694.449,A -85,B 0,C 180,E1 -20776.42,E2 -20776.42} C_VEL
LIN {X 0,Y 226.058,Z 681.825,A -85,B 0,C 180,E1 -20777.661,E2 -20777.661} C_VEL
LIN {X 0,Y 227.216,Z 669.347,A -85,B 0,C 180,E1 -20778.546,E2 -20778.546} C_VEL
LIN {X 0,Y 228.072,Z 655.645,A -85,B 0,C 180,E1 -20779.151,E2 -20779.151} C_VEL
LIN {X 0,Y 230.629,Z 599.368,A -85,B 0,C 180,E1 -20781.035,E2 -20781.035} C_VEL
LIN {X 0,Y 223.899,Z 580.724,A -85,B 0,C 180,E1 -20782.573,E2 -20782.573} C_VEL
LIN {X 0,Y 218.254,Z 566.672,A -85,B 0,C 180,E1 -20783.869,E2 -20783.869} C_VEL
LIN {X 0,Y 214.317,Z 558.874,A -85,B 0,C 180,E1 -20784.74,E2 -20784.74} C_VEL
LIN {X 0,Y 214.12,Z 557.816,A -85,B 0,C 180,E1 -20784.824,E2 -20784.824} C_VEL
LIN {X 0,Y 214.444,Z 557.773,A -85,B 0,C 180,E1 -20788.125,E2 -20788.125} C_VEL
LIN {X 0,Y 214.548,Z 557.761,A -85,B 0,C 180,E1 -20790.003,E2 -20790.003} C_VEL
LIN {X 0,Y 214.444,Z 557.771,A -85,B 0,C 180,E1 -20791.881,E2 -20791.881} C_VEL
LIN {X 0,Y 214.238,Z 557.8,A -85,B 0,C 180,E1 -20797.543,E2 -20797.543} C_VEL
LIN {X 0,Y 214.044,Z 557.815,A -85,B 0,C 180,E1 -20801.365,E2 -20801.365} C_VEL
LIN {X 0,Y 213.934,Z 557.834,A -85,B 0,C 180,E1 -20805.24,E2 -20805.24} C_VEL
LIN {X 0,Y 213.933,Z 557.835,A -85,B 0,C 180,E1 -20807.698,E2 -20807.698} C_VEL
LIN {X 0,Y 213.848,Z 557.826,A -85,B 0,C 180,E1 -20813.23,E2 -20813.23} C_VEL
LIN {X 0,Y 213.831,Z 557.852,A -85,B 0,C 180,E1 -20817.452,E2 -20817.452} C_VEL
LIN {X 0,Y 213.769,Z 557.85,A -85,B 0,C 180,E1 -20821.74,E2 -20821.74} C_VEL
LIN {X 0,Y 213.746,Z 557.86,A -85,B 0,C 180,E1 -20826.291,E2 -20826.291} C_VEL
LIN {X 0,Y 213.716,Z 557.855,A -85,B 0,C 180,E1 -20831.128,E2 -20831.128} C_VEL
LIN {X 0,Y 213.711,Z 557.864,A -85,B 0,C 180,E1 -20833.68,E2 -20833.68} C_VEL
LIN {X 0,Y 213.711,Z 557.862,A -85,B 0,C 180,E1 -20836.346,E2 -20836.346} C_VEL
LIN {X 0,Y 213.722,Z 557.855,A -85,B 0,C 180,E1 -20839.145,E2 -20839.145} C_VEL
LIN {X 0,Y 213.749,Z 557.859,A -85,B 0,C 180,E1 -20843.714,E2 -20843.714} C_VEL
LIN {X 0,Y 213.801,Z 557.848,A -85,B 0,C 180,E1 -20848.727,E2 -20848.727} C_VEL
LIN {X 0,Y 213.833,Z 557.838,A -85,B 0,C 180,E1 -20852.605,E2 -20852.605} C_VEL
LIN {X 0,Y 213.826,Z 557.848,A -85,B 0,C 180,E1 -20856.976,E2 -20856.976} C_VEL
LIN {X 0,Y 213.928,Z 557.82,A -85,B 0,C 180,E1 -20862.803,E2 -20862.803} C_VEL
LIN {X 0,Y 213.952,Z 557.831,A -85,B 0,C 180,E1 -20866.707,E2 -20866.707} C_VEL
LIN {X 0,Y 214.15,Z 557.804,A -85,B 0,C 180,E1 -20870.557,E2 -20870.557} C_VEL
LIN {X 0,Y 214.108,Z 557.805,A -85,B 0,C 180,E1 -20874.35,E2 -20874.35} C_VEL
LIN {X 0,Y 214.454,Z 557.772,A -85,B 0,C 180,E1 -20878.123,E2 -20878.123} C_VEL
LIN {X 0,Y 214.559,Z 557.758,A -85,B 0,C 180,E1 -20880.001,E2 -20880.001} C_VEL
LIN {X 0,Y 214.454,Z 557.766,A -85,B 0,C 180,E1 -20881.879,E2 -20881.879} C_VEL
LIN {X 0,Y 214.257,Z 557.795,A -85,B 0,C 180,E1 -20887.54,E2 -20887.54} C_VEL
LIN {X 0,Y 214.052,Z 557.819,A -85,B 0,C 180,E1 -20891.362,E2 -20891.362} C_VEL
LIN {X 0,Y 213.943,Z 557.833,A -85,B 0,C 180,E1 -20895.237,E2 -20895.237} C_VEL
LIN {X 0,Y 213.846,Z 557.845,A -85,B 0,C 180,E1 -20899.188,E2 -20899.188} C_VEL
LIN {X 0,Y 213.821,Z 557.827,A -85,B 0,C 180,E1 -20903.231,E2 -20903.231} C_VEL
LIN {X 0,Y 213.839,Z 557.841,A -85,B 0,C 180,E1 -20907.45,E2 -20907.45} C_VEL
LIN {X 0,Y 213.778,Z 557.855,A -85,B 0,C 180,E1 -20911.737,E2 -20911.737} C_VEL
LIN {X 0,Y 213.754,Z 557.859,A -85,B 0,C 180,E1 -20916.287,E2 -20916.287} C_VEL
LIN {X 0,Y 213.721,Z 557.862,A -85,B 0,C 180,E1 -20921.124,E2 -20921.124} C_VEL
LIN {X 0,Y 213.713,Z 557.864,A -85,B 0,C 180,E1 -20923.678,E2 -20923.678} C_VEL
LIN {X 0,Y 213.712,Z 557.861,A -85,B 0,C 180,E1 -20926.344,E2 -20926.344} C_VEL
LIN {X 0,Y 213.785,Z 557.855,A -85,B 0,C 180,E1 -20930.383,E2 -20930.383} C_VEL
LIN {X 0,Y 213.564,Z 558.609,A -85,B 0,C 180,E1 -20931.139,E2 -20931.139} C_VEL
LIN {X 0,Y 212.173,Z 561.812,A -85,B 0,C 180,E1 -20932.456,E2 -20932.456} C_VEL
LIN {X 0,Y 210.611,Z 565.118,A -85,B 0,C 180,E1 -20933.568,E2 -20933.568} C_VEL
LIN {X 0,Y 209.92,Z 568.466,A -85,B 0,C 180,E1 -20934.373,E2 -20934.373} C_VEL
LIN {X 0,Y 210.279,Z 571.239,A -85,B 0,C 180,E1 -20934.76,E2 -20934.76} C_VEL
LIN {X 0,Y 219.506,Z 595.061,A -85,B 0,C 180,E1 -20937.005,E2 -20937.005} C_VEL
LIN {X 0,Y 220.68,Z 598.704,A -85,B 0,C 180,E1 -20937.299,E2 -20937.299} C_VEL
LIN {X 0,Y 223.474,Z 620.684,A -85,B 0,C 180,E1 -20938.519,E2 -20938.519} C_VEL
LIN {X 0,Y 220.867,Z 676.435,A -85,B 0,C 180,E1 -20940.511,E2 -20940.511} C_VEL
LIN {X 0,Y 219.586,Z 689.517,A -85,B 0,C 180,E1 -20941.306,E2 -20941.306} C_VEL
LIN {X 0,Y 217.98,Z 701.708,A -85,B 0,C 180,E1 -20942.386,E2 -20942.386} C_VEL
LIN {X 0,Y 216.249,Z 712.783,A -85,B 0,C 180,E1 -20943.714,E2 -20943.714} C_VEL
LIN {X 0,Y 214.187,Z 724.402,A -85,B 0,C 180,E1 -20945.525,E2 -20945.525} C_VEL
LIN {X 0,Y 212.227,Z 733.799,A -85,B 0,C 180,E1 -20947.356,E2 -20947.356} C_VEL
LIN {X 0,Y 210.126,Z 743.32,A -85,B 0,C 180,E1 -20949.654,E2 -20949.654} C_VEL
LIN {X 0,Y 208.62,Z 750.641,A -85,B 0,C 180,E1 -20951.841,E2 -20951.841} C_VEL
LIN {X 0,Y 206.926,Z 758.502,A -85,B 0,C 180,E1 -20954.736,E2 -20954.736} C_VEL
LIN {X 0,Y 205.844,Z 763.853,A -85,B 0,C 180,E1 -20957.175,E2 -20957.175} C_VEL
LIN {X 0,Y 205.046,Z 769.016,A -85,B 0,C 180,E1 -20960.129,E2 -20960.129} C_VEL
LIN {X 0,Y 204.568,Z 772.983,A -85,B 0,C 180,E1 -20963.091,E2 -20963.091} C_VEL
LIN {X 0,Y 204.368,Z 775.87,A -85,B 0,C 180,E1 -20966.053,E2 -20966.053} C_VEL
LIN {X 0,Y 204.401,Z 777.217,A -85,B 0,C 180,E1 -20968.027,E2 -20968.027} C_VEL
LIN {X 0,Y 204.499,Z 778.153,A -85,B 0,C 180,E1 -20969.997,E2 -20969.997} C_VEL
LIN {X 0,Y 204.358,Z 778.675,A -85,B 0,C 180,E1 -20971.968,E2 -20971.968} C_VEL
LIN {X 0,Y 204.323,Z 778.755,A -85,B 0,C 180,E1 -20974.042,E2 -20974.042} C_VEL
LIN {X 0,Y 204.645,Z 777.741,A -85,B 0,C 180,E1 -20977.893,E2 -20977.893} C_VEL
LIN {X 0,Y 205.077,Z 776.648,A -85,B 0,C 180,E1 -20979.863,E2 -20979.863} C_VEL
LIN {X 0,Y 205.707,Z 775.13,A -85,B 0,C 180,E1 -20981.826,E2 -20981.826} C_VEL
LIN {X 0,Y 206.965,Z 772.071,A -85,B 0,C 180,E1 -20984.752,E2 -20984.752} C_VEL
LIN {X 0,Y 208.916,Z 767.977,A -85,B 0,C 180,E1 -20987.621,E2 -20987.621} C_VEL
LIN {X 0,Y 211.806,Z 761.736,A -85,B 0,C 180,E1 -20990.895,E2 -20990.895} C_VEL
LIN {X 0,Y 214.594,Z 754.995,A -85,B 0,C 180,E1 -20993.649,E2 -20993.649} C_VEL
LIN {X 0,Y 218.089,Z 746.671,A -85,B 0,C 180,E1 -20996.299,E2 -20996.299} C_VEL
LIN {X 0,Y 221.382,Z 738.217,A -85,B 0,C 180,E1 -20998.434,E2 -20998.434} C_VEL
LIN {X 0,Y 224.957,Z 727.875,A -85,B 0,C 180,E1 -21000.506,E2 -21000.506} C_VEL
LIN {X 0,Y 228.554,Z 716.325,A -85,B 0,C 180,E1 -21002.292,E2 -21002.292} C_VEL
LIN {X 0,Y 231.479,Z 704.955,A -85,B 0,C 180,E1 -21003.645,E2 -21003.645} C_VEL
LIN {X 0,Y 234.157,Z 692.178,A -85,B 0,C 180,E1 -21004.765,E2 -21004.765} C_VEL
LIN {X 0,Y 236.219,Z 679.359,A -85,B 0,C 180,E1 -21005.547,E2 -21005.547} C_VEL
LIN {X 0,Y 237.544,Z 664.496,A -85,B 0,C 180,E1 -21006.137,E2 -21006.137} C_VEL
LIN {X 0,Y 240.204,Z 624.674,A -85,B 0,C 180,E1 -21007.473,E2 -21007.473} C_VEL
LIN {X 0,Y 239.487,Z 618.037,A -85,B 0,C 180,E1 -21008,E2 -21008} C_VEL
LIN {X 0,Y 234.964,Z 607.333,A -85,B 0,C 180,E1 -21009.807,E2 -21009.807} C_VEL
LIN {X 0,Y 230.03,Z 596.979,A -85,B 0,C 180,E1 -21011.921,E2 -21011.921} C_VEL
LIN {X 0,Y 226.277,Z 590.443,A -85,B 0,C 180,E1 -21013.601,E2 -21013.601} C_VEL
LIN {X 0,Y 224.298,Z 587.058,A -85,B 0,C 180,E1 -21014.565,E2 -21014.565} C_VEL
LIN {X 0,Y 220.938,Z 581.693,A -85,B 0,C 180,E1 -21016.286,E2 -21016.286} C_VEL
LIN {X 0,Y 217.898,Z 576.85,A -85,B 0,C 180,E1 -21018.009,E2 -21018.009} C_VEL
LIN {X 0,Y 213.851,Z 571.301,A -85,B 0,C 180,E1 -21020.526,E2 -21020.526} C_VEL
LIN {X 0,Y 212.827,Z 569.892,A -85,B 0,C 180,E1 -21021.239,E2 -21021.239} C_VEL
LIN {X 0,Y 209.617,Z 565.818,A -85,B 0,C 180,E1 -21023.68,E2 -21023.68} C_VEL
LIN {X 0,Y 208.285,Z 563.555,A -85,B 0,C 180,E1 -21024.996,E2 -21024.996} C_VEL
LIN {X 0,Y 207.73,Z 561.533,A -85,B 0,C 180,E1 -21027.753,E2 -21027.753} C_VEL
LIN {X 0,Y 206.748,Z 558.722,A -85,B 0,C 180,E1 -21033.34,E2 -21033.34} C_VEL
LIN {X 0,Y 206.75,Z 558.728,A -85,B 0,C 180,E1 -21038.041,E2 -21038.041} C_VEL
LIN {X 0,Y 206.864,Z 558.717,A -85,B 0,C 180,E1 -21042.195,E2 -21042.195} C_VEL
LIN {X 0,Y 206.905,Z 558.714,A -85,B 0,C 180,E1 -21046.244,E2 -21046.244} C_VEL
LIN {X 0,Y 207.154,Z 558.672,A -85,B 0,C 180,E1 -21051.217,E2 -21051.217} C_VEL
LIN {X 0,Y 207.401,Z 560.111,A -85,B 0,C 180,E1 -21054.408,E2 -21054.408} C_VEL
LIN {X 0,Y 208.859,Z 562.582,A -85,B 0,C 180,E1 -21055.899,E2 -21055.899} C_VEL
LIN {X 0,Y 212.877,Z 566.151,A -85,B 0,C 180,E1 -21058.935,E2 -21058.935} C_VEL
LIN {X 0,Y 217.358,Z 572.187,A -85,B 0,C 180,E1 -21061.852,E2 -21061.852} C_VEL
LIN {X 0,Y 220.337,Z 576.407,A -85,B 0,C 180,E1 -21063.571,E2 -21063.571} C_VEL
LIN {X 0,Y 224.576,Z 582.5,A -85,B 0,C 180,E1 -21065.728,E2 -21065.728} C_VEL
LIN {X 0,Y 229.595,Z 590.79,A -85,B 0,C 180,E1 -21068.058,E2 -21068.058} C_VEL
LIN {X 0,Y 235.076,Z 600.888,A -85,B 0,C 180,E1 -21070.37,E2 -21070.37} C_VEL
LIN {X 0,Y 239.428,Z 610.259,A -85,B 0,C 180,E1 -21072.075,E2 -21072.075} C_VEL
LIN {X 0,Y 240.895,Z 614.137,A -85,B 0,C 180,E1 -21072.661,E2 -21072.661} C_VEL
LIN {X 0,Y 237.181,Z 665.479,A -85,B 0,C 180,E1 -21074.391,E2 -21074.391} C_VEL
LIN {X 0,Y 235.512,Z 678.564,A -85,B 0,C 180,E1 -21075.121,E2 -21075.121} C_VEL
LIN {X 0,Y 233.478,Z 690.026,A -85,B 0,C 180,E1 -21076.04,E2 -21076.04} C_VEL
LIN {X 0,Y 230.652,Z 702.488,A -85,B 0,C 180,E1 -21077.398,E2 -21077.398} C_VEL
LIN {X 0,Y 227.612,Z 713.439,A -85,B 0,C 180,E1 -21078.969,E2 -21078.969} C_VEL
LIN {X 0,Y 224.503,Z 723.269,A -85,B 0,C 180,E1 -21080.768,E2 -21080.768} C_VEL
LIN {X 0,Y 221.13,Z 732.386,A -85,B 0,C 180,E1 -21082.834,E2 -21082.834} C_VEL
LIN {X 0,Y 217.646,Z 740.915,A -85,B 0,C 180,E1 -21085.299,E2 -21085.299} C_VEL
LIN {X 0,Y 214.192,Z 748.726,A -85,B 0,C 180,E1 -21088.183,E2 -21088.183} C_VEL
LIN {X 0,Y 211.14,Z 755.174,A -85,B 0,C 180,E1 -21091.299,E2 -21091.299} C_VEL
LIN {X 0,Y 209.034,Z 759.366,A -85,B 0,C 180,E1 -21093.96,E2 -21093.96} C_VEL
LIN {X 0,Y 207.87,Z 761.624,A -85,B 0,C 180,E1 -21095.77,E2 -21095.77} C_VEL
LIN {X 0,Y 206.48,Z 764.263,A -85,B 0,C 180,E1 -21098.482,E2 -21098.482} C_VEL
LIN {X 0,Y 205.434,Z 766.024,A -85,B 0,C 180,E1 -21101.186,E2 -21101.186} C_VEL
LIN {X 0,Y 204.687,Z 767.018,A -85,B 0,C 180,E1 -21103.864,E2 -21103.864} C_VEL
LIN {X 0,Y 204.219,Z 767.297,A -85,B 0,C 180,E1 -21106.51,E2 -21106.51} C_VEL
LIN {X 0,Y 203.971,Z 766.785,A -85,B 0,C 180,E1 -21109.289,E2 -21109.289} C_VEL
LIN {X 0,Y 204.012,Z 765.264,A -85,B 0,C 180,E1 -21112.401,E2 -21112.401} C_VEL
LIN {X 0,Y 204.412,Z 762.614,A -85,B 0,C 180,E1 -21115.603,E2 -21115.603} C_VEL
LIN {X 0,Y 205.162,Z 758.337,A -85,B 0,C 180,E1 -21119.084,E2 -21119.084} C_VEL
LIN {X 0,Y 206.24,Z 752.811,A -85,B 0,C 180,E1 -21122.372,E2 -21122.372} C_VEL
LIN {X 0,Y 207.665,Z 746.062,A -85,B 0,C 180,E1 -21125.47,E2 -21125.47} C_VEL
LIN {X 0,Y 209.457,Z 738.039,A -85,B 0,C 180,E1 -21128.344,E2 -21128.344} C_VEL
LIN {X 0,Y 211.607,Z 728.273,A -85,B 0,C 180,E1 -21131.109,E2 -21131.109} C_VEL
LIN {X 0,Y 213.695,Z 718.186,A -85,B 0,C 180,E1 -21133.365,E2 -21133.365} C_VEL
LIN {X 0,Y 215.971,Z 706.061,A -85,B 0,C 180,E1 -21135.485,E2 -21135.485} C_VEL
LIN {X 0,Y 217.786,Z 694.383,A -85,B 0,C 180,E1 -21137.066,E2 -21137.066} C_VEL
LIN {X 0,Y 219.463,Z 681.705,A -85,B 0,C 180,E1 -21138.34,E2 -21138.34} C_VEL
LIN {X 0,Y 220.727,Z 668.452,A -85,B 0,C 180,E1 -21139.288,E2 -21139.288} C_VEL
LIN {X 0,Y 221.663,Z 653.254,A -85,B 0,C 180,E1 -21139.932,E2 -21139.932} C_VEL
LIN {X 0,Y 223.972,Z 600.455,A -85,B 0,C 180,E1 -21141.773,E2 -21141.773} C_VEL
LIN {X 0,Y 216.532,Z 579.997,A -85,B 0,C 180,E1 -21143.539,E2 -21143.539} C_VEL
LIN {X 0,Y 212.349,Z 569.777,A -85,B 0,C 180,E1 -21144.547,E2 -21144.547} C_VEL
LIN {X 0,Y 207.305,Z 559.758,A -85,B 0,C 180,E1 -21145.72,E2 -21145.72} C_VEL
LIN {X 0,Y 207.08,Z 558.696,A -85,B 0,C 180,E1 -21145.867,E2 -21145.867} C_VEL
LIN {X 0,Y 207.38,Z 558.653,A -85,B 0,C 180,E1 -21148.061,E2 -21148.061} C_VEL
LIN {X 0,Y 207.513,Z 558.637,A -85,B 0,C 180,E1 -21150.003,E2 -21150.003} C_VEL
LIN {X 0,Y 207.38,Z 558.651,A -85,B 0,C 180,E1 -21151.945,E2 -21151.945} C_VEL
LIN {X 0,Y 207.176,Z 558.679,A -85,B 0,C 180,E1 -21157.801,E2 -21157.801} C_VEL
LIN {X 0,Y 206.981,Z 558.693,A -85,B 0,C 180,E1 -21161.758,E2 -21161.758} C_VEL
LIN {X 0,Y 206.872,Z 558.715,A -85,B 0,C 180,E1 -21165.773,E2 -21165.773} C_VEL
LIN {X 0,Y 206.784,Z 558.718,A -85,B 0,C 180,E1 -21169.872,E2 -21169.872} C_VEL
LIN {X 0,Y 206.765,Z 558.716,A -85,B 0,C 180,E1 -21174.075,E2 -21174.075} C_VEL
LIN {X 0,Y 206.738,Z 558.733,A -85,B 0,C 180,E1 -21178.422,E2 -21178.422} C_VEL
LIN {X 0,Y 206.701,Z 558.73,A -85,B 0,C 180,E1 -21182.96,E2 -21182.96} C_VEL
LIN {X 0,Y 206.682,Z 558.739,A -85,B 0,C 180,E1 -21187.742,E2 -21187.742} C_VEL
LIN {X 0,Y 206.646,Z 558.736,A -85,B 0,C 180,E1 -21191.565,E2 -21191.565} C_VEL
LIN {X 0,Y 206.639,Z 558.746,A -85,B 0,C 180,E1 -21195.584,E2 -21195.584} C_VEL
LIN {X 0,Y 206.665,Z 558.728,A -85,B 0,C 180,E1 -21199.751,E2 -21199.751} C_VEL
LIN {X 0,Y 206.704,Z 558.735,A -85,B 0,C 180,E1 -21204.691,E2 -21204.691} C_VEL
LIN {X 0,Y 206.729,Z 558.726,A -85,B 0,C 180,E1 -21209.341,E2 -21209.341} C_VEL
LIN {X 0,Y 206.738,Z 558.727,A -85,B 0,C 180,E1 -21213.774,E2 -21213.774} C_VEL
LIN {X 0,Y 206.742,Z 558.73,A -85,B 0,C 180,E1 -21218.043,E2 -21218.043} C_VEL
LIN {X 0,Y 206.875,Z 558.699,A -85,B 0,C 180,E1 -21222.198,E2 -21222.198} C_VEL
LIN {X 0,Y 206.892,Z 558.711,A -85,B 0,C 180,E1 -21226.245,E2 -21226.245} C_VEL
LIN {X 0,Y 207.108,Z 558.682,A -85,B 0,C 180,E1 -21230.232,E2 -21230.232} C_VEL
LIN {X 0,Y 207.069,Z 558.679,A -85,B 0,C 180,E1 -21234.157,E2 -21234.157} C_VEL
LIN {X 0,Y 207.39,Z 558.652,A -85,B 0,C 180,E1 -21238.059,E2 -21238.059} C_VEL
LIN {X 0,Y 207.524,Z 558.634,A -85,B 0,C 180,E1 -21240.001,E2 -21240.001} C_VEL
LIN {X 0,Y 207.391,Z 558.645,A -85,B 0,C 180,E1 -21241.943,E2 -21241.943} C_VEL
LIN {X 0,Y 207.198,Z 558.676,A -85,B 0,C 180,E1 -21247.799,E2 -21247.799} C_VEL
LIN {X 0,Y 206.985,Z 558.696,A -85,B 0,C 180,E1 -21251.756,E2 -21251.756} C_VEL
LIN {X 0,Y 206.877,Z 558.715,A -85,B 0,C 180,E1 -21255.771,E2 -21255.771} C_VEL
LIN {X 0,Y 206.788,Z 558.722,A -85,B 0,C 180,E1 -21259.87,E2 -21259.87} C_VEL
LIN {X 0,Y 206.757,Z 558.703,A -85,B 0,C 180,E1 -21264.074,E2 -21264.074} C_VEL
LIN {X 0,Y 206.747,Z 558.731,A -85,B 0,C 180,E1 -21268.419,E2 -21268.419} C_VEL
LIN {X 0,Y 206.71,Z 558.735,A -85,B 0,C 180,E1 -21272.957,E2 -21272.957} C_VEL
LIN {X 0,Y 206.69,Z 558.74,A -85,B 0,C 180,E1 -21277.739,E2 -21277.739} C_VEL
LIN {X 0,Y 206.651,Z 558.744,A -85,B 0,C 180,E1 -21281.562,E2 -21281.562} C_VEL
LIN {X 0,Y 206.64,Z 558.739,A -85,B 0,C 180,E1 -21285.581,E2 -21285.581} C_VEL
LIN {X 0,Y 206.745,Z 558.814,A -85,B 0,C 180,E1 -21290.256,E2 -21290.256} C_VEL
LIN {X 0,Y 208.678,Z 567.12,A -85,B 0,C 180,E1 -21294.349,E2 -21294.349} C_VEL
LIN {X 0,Y 210.279,Z 571.239,A -85,B 0,C 180,E1 -21294.76,E2 -21294.76} C_VEL
LIN {X 0,Y 211.973,Z 578.662,A -85,B 0,C 180,E1 -21295.32,E2 -21295.32} C_VEL
LIN {X 0,Y 214.501,Z 601.791,A -85,B 0,C 180,E1 -21296.653,E2 -21296.653} C_VEL
LIN {X 0,Y 216.947,Z 621.337,A -85,B 0,C 180,E1 -21297.778,E2 -21297.778} C_VEL
LIN {X 0,Y 214.321,Z 676.004,A -85,B 0,C 180,E1 -21299.788,E2 -21299.788} C_VEL
LIN {X 0,Y 213.001,Z 689.147,A -85,B 0,C 180,E1 -21300.604,E2 -21300.604} C_VEL
LIN {X 0,Y 211.357,Z 701.383,A -85,B 0,C 180,E1 -21301.714,E2 -21301.714} C_VEL
LIN {X 0,Y 209.568,Z 712.49,A -85,B 0,C 180,E1 -21303.078,E2 -21303.078} C_VEL
LIN {X 0,Y 207.43,Z 724.125,A -85,B 0,C 180,E1 -21304.94,E2 -21304.94} C_VEL
LIN {X 0,Y 205.21,Z 734.626,A -85,B 0,C 180,E1 -21307.069,E2 -21307.069} C_VEL
LIN {X 0,Y 203.195,Z 743.192,A -85,B 0,C 180,E1 -21309.229,E2 -21309.229} C_VEL
LIN {X 0,Y 201.484,Z 751.132,A -85,B 0,C 180,E1 -21311.701,E2 -21311.701} C_VEL
LIN {X 0,Y 199.77,Z 758.839,A -85,B 0,C 180,E1 -21314.698,E2 -21314.698} C_VEL
LIN {X 0,Y 198.537,Z 765.017,A -85,B 0,C 180,E1 -21317.734,E2 -21317.734} C_VEL
LIN {X 0,Y 197.809,Z 769.885,A -85,B 0,C 180,E1 -21320.797,E2 -21320.797} C_VEL
LIN {X 0,Y 197.411,Z 773.577,A -85,B 0,C 180,E1 -21323.866,E2 -21323.866} C_VEL
LIN {X 0,Y 197.289,Z 775.463,A -85,B 0,C 180,E1 -21325.912,E2 -21325.912} C_VEL
LIN {X 0,Y 197.305,Z 776.863,A -85,B 0,C 180,E1 -21327.956,E2 -21327.956} C_VEL
LIN {X 0,Y 197.416,Z 777.842,A -85,B 0,C 180,E1 -21329.997,E2 -21329.997} C_VEL
LIN {X 0,Y 197.245,Z 778.567,A -85,B 0,C 180,E1 -21333.906,E2 -21333.906} C_VEL
LIN {X 0,Y 197.343,Z 778.3,A -85,B 0,C 180,E1 -21336.13,E2 -21336.13} C_VEL
LIN {X 0,Y 198.054,Z 776.595,A -85,B 0,C 180,E1 -21340.217,E2 -21340.217} C_VEL
LIN {X 0,Y 198.724,Z 775.158,A -85,B 0,C 180,E1 -21342.248,E2 -21342.248} C_VEL
LIN {X 0,Y 200.088,Z 772.172,A -85,B 0,C 180,E1 -21345.271,E2 -21345.271} C_VEL
LIN {X 0,Y 202.154,Z 768.172,A -85,B 0,C 180,E1 -21348.23,E2 -21348.23} C_VEL
LIN {X 0,Y 204.747,Z 763.058,A -85,B 0,C 180,E1 -21351.123,E2 -21351.123} C_VEL
LIN {X 0,Y 207.612,Z 756.726,A -85,B 0,C 180,E1 -21353.964,E2 -21353.964} C_VEL
LIN {X 0,Y 211.147,Z 748.85,A -85,B 0,C 180,E1 -21356.698,E2 -21356.698} C_VEL
LIN {X 0,Y 215.222,Z 739.107,A -85,B 0,C 180,E1 -21359.325,E2 -21359.325} C_VEL
LIN {X 0,Y 218.957,Z 729.066,A -85,B 0,C 180,E1 -21361.435,E2 -21361.435} C_VEL
LIN {X 0,Y 222.667,Z 717.806,A -85,B 0,C 180,E1 -21363.254,E2 -21363.254} C_VEL
LIN {X 0,Y 226.153,Z 705.173,A -85,B 0,C 180,E1 -21364.819,E2 -21364.819} C_VEL
LIN {X 0,Y 228.931,Z 692.611,A -85,B 0,C 180,E1 -21365.95,E2 -21365.95} C_VEL
LIN {X 0,Y 231.161,Z 679.576,A -85,B 0,C 180,E1 -21366.763,E2 -21366.763} C_VEL
LIN {X 0,Y 232.553,Z 665.242,A -85,B 0,C 180,E1 -21367.355,E2 -21367.355} C_VEL
LIN {X 0,Y 235.334,Z 625.526,A -85,B 0,C 180,E1 -21368.717,E2 -21368.717} C_VEL
LIN {X 0,Y 234.834,Z 621.262,A -85,B 0,C 180,E1 -21369.083,E2 -21369.083} C_VEL
LIN {X 0,Y 230.121,Z 609.808,A -85,B 0,C 180,E1 -21371.122,E2 -21371.122} C_VEL
LIN {X 0,Y 225.984,Z 601.178,A -85,B 0,C 180,E1 -21373.02,E2 -21373.02} C_VEL
LIN {X 0,Y 221.618,Z 593.167,A -85,B 0,C 180,E1 -21375.195,E2 -21375.195} C_VEL
LIN {X 0,Y 217.856,Z 587.118,A -85,B 0,C 180,E1 -21377.216,E2 -21377.216} C_VEL
LIN {X 0,Y 214.75,Z 582.125,A -85,B 0,C 180,E1 -21379.115,E2 -21379.115} C_VEL
LIN {X 0,Y 211.294,Z 576.935,A -85,B 0,C 180,E1 -21381.462,E2 -21381.462} C_VEL
LIN {X 0,Y 207.635,Z 572.133,A -85,B 0,C 180,E1 -21384.372,E2 -21384.372} C_VEL
LIN {X 0,Y 206.171,Z 569.912,A -85,B 0,C 180,E1 -21385.773,E2 -21385.773} C_VEL
LIN {X 0,Y 200.781,Z 562.61,A -85,B 0,C 180,E1 -21393.072,E2 -21393.072} C_VEL
LIN {X 0,Y 200.224,Z 561.453,A -85,B 0,C 180,E1 -21397.286,E2 -21397.286} C_VEL
LIN {X 0,Y 200.057,Z 560.91,A -85,B 0,C 180,E1 -21401.567,E2 -21401.567} C_VEL
LIN {X 0,Y 200.295,Z 561.298,A -85,B 0,C 180,E1 -21406.299,E2 -21406.299} C_VEL
LIN {X 0,Y 202.426,Z 564.011,A -85,B 0,C 180,E1 -21410.161,E2 -21410.161} C_VEL
LIN {X 0,Y 204.13,Z 565.461,A -85,B 0,C 180,E1 -21412.332,E2 -21412.332} C_VEL
LIN {X 0,Y 205.776,Z 567.153,A -85,B 0,C 180,E1 -21414.05,E2 -21414.05} C_VEL
LIN {X 0,Y 207.67,Z 569.758,A -85,B 0,C 180,E1 -21415.875,E2 -21415.875} C_VEL
LIN {X 0,Y 210.912,Z 572.724,A -85,B 0,C 180,E1 -21418.388,E2 -21418.388} C_VEL
LIN {X 0,Y 214.919,Z 578.395,A -85,B 0,C 180,E1 -21421.155,E2 -21421.155} C_VEL
LIN {X 0,Y 219.012,Z 584.375,A -85,B 0,C 180,E1 -21423.592,E2 -21423.592} C_VEL
LIN {X 0,Y 221.746,Z 588.44,A -85,B 0,C 180,E1 -21425.024,E2 -21425.024} C_VEL
LIN {X 0,Y 227.404,Z 598.262,A -85,B 0,C 180,E1 -21427.784,E2 -21427.784} C_VEL
LIN {X 0,Y 231.965,Z 607.186,A -85,B 0,C 180,E1 -21429.797,E2 -21429.797} C_VEL
LIN {X 0,Y 235.91,Z 616.291,A -85,B 0,C 180,E1 -21431.445,E2 -21431.445} C_VEL
LIN {X 0,Y 232.188,Z 666.135,A -85,B 0,C 180,E1 -21433.176,E2 -21433.176} C_VEL
LIN {X 0,Y 230.455,Z 678.768,A -85,B 0,C 180,E1 -21433.886,E2 -21433.886} C_VEL
LIN {X 0,Y 228.059,Z 691.626,A -85,B 0,C 180,E1 -21434.956,E2 -21434.956} C_VEL
LIN {X 0,Y 225.127,Z 703.573,A -85,B 0,C 180,E1 -21436.317,E2 -21436.317} C_VEL
LIN {X 0,Y 221.713,Z 715.087,A -85,B 0,C 180,E1 -21438.028,E2 -21438.028} C_VEL
LIN {X 0,Y 218.105,Z 725.644,A -85,B 0,C 180,E1 -21440.074,E2 -21440.074} C_VEL
LIN {X 0,Y 214.311,Z 735.092,A -85,B 0,C 180,E1 -21442.394,E2 -21442.394} C_VEL
LIN {X 0,Y 210.804,Z 743.113,A -85,B 0,C 180,E1 -21444.905,E2 -21444.905} C_VEL
LIN {X 0,Y 207.644,Z 749.673,A -85,B 0,C 180,E1 -21447.497,E2 -21447.497} C_VEL
LIN {X 0,Y 204.402,Z 755.958,A -85,B 0,C 180,E1 -21450.737,E2 -21450.737} C_VEL
LIN {X 0,Y 201.955,Z 760.468,A -85,B 0,C 180,E1 -21453.833,E2 -21453.833} C_VEL
LIN {X 0,Y 200.268,Z 763.476,A -85,B 0,C 180,E1 -21456.624,E2 -21456.624} C_VEL
LIN {X 0,Y 198.924,Z 765.659,A -85,B 0,C 180,E1 -21459.488,E2 -21459.488} C_VEL
LIN {X 0,Y 197.922,Z 766.999,A -85,B 0,C 180,E1 -21462.427,E2 -21462.427} C_VEL
LIN {X 0,Y 197.278,Z 767.498,A -85,B 0,C 180,E1 -21465.437,E2 -21465.437} C_VEL
LIN {X 0,Y 196.895,Z 767.114,A -85,B 0,C 180,E1 -21468.552,E2 -21468.552} C_VEL
LIN {X 0,Y 196.936,Z 765.203,A -85,B 0,C 180,E1 -21472.655,E2 -21472.655} C_VEL
LIN {X 0,Y 197.472,Z 761.788,A -85,B 0,C 180,E1 -21476.524,E2 -21476.524} C_VEL
LIN {X 0,Y 198.137,Z 758.224,A -85,B 0,C 180,E1 -21479.369,E2 -21479.369} C_VEL
LIN {X 0,Y 199.252,Z 752.72,A -85,B 0,C 180,E1 -21482.711,E2 -21482.711} C_VEL
LIN {X 0,Y 200.589,Z 746.54,A -85,B 0,C 180,E1 -21485.635,E2 -21485.635} C_VEL
LIN {X 0,Y 202.294,Z 739.122,A -85,B 0,C 180,E1 -21488.438,E2 -21488.438} C_VEL
LIN {X 0,Y 204.386,Z 729.909,A -85,B 0,C 180,E1 -21491.197,E2 -21491.197} C_VEL
LIN {X 0,Y 206.517,Z 720.041,A -85,B 0,C 180,E1 -21493.558,E2 -21493.558} C_VEL
LIN {X 0,Y 208.721,Z 709.104,A -85,B 0,C 180,E1 -21495.624,E2 -21495.624} C_VEL
LIN {X 0,Y 210.861,Z 696.332,A -85,B 0,C 180,E1 -21497.491,E2 -21497.491} C_VEL
LIN {X 0,Y 212.63,Z 683.958,A -85,B 0,C 180,E1 -21498.836,E2 -21498.836} C_VEL
LIN {X 0,Y 214.041,Z 669.909,A -85,B 0,C 180,E1 -21499.915,E2 -21499.915} C_VEL
LIN {X 0,Y 214.979,Z 656.379,A -85,B 0,C 180,E1 -21500.552,E2 -21500.552} C_VEL
LIN {X 0,Y 217.5,Z 602.069,A -85,B 0,C 180,E1 -21502.495,E2 -21502.495} C_VEL
LIN {X 0,Y 210.812,Z 583.498,A -85,B 0,C 180,E1 -21504.167,E2 -21504.167} C_VEL
LIN {X 0,Y 206.605,Z 573.162,A -85,B 0,C 180,E1 -21505.221,E2 -21505.221} C_VEL
LIN {X 0,Y 200.334,Z 560.632,A -85,B 0,C 180,E1 -21506.735,E2 -21506.735} C_VEL
LIN {X 0,Y 200.133,Z 559.558,A -85,B 0,C 180,E1 -21506.858,E2 -21506.858} C_VEL
LIN {X 0,Y 200.477,Z 559.513,A -85,B 0,C 180,E1 -21510.003,E2 -21510.003} C_VEL
LIN {X 0,Y 200.03,Z 559.566,A -85,B 0,C 180,E1 -21514.032,E2 -21514.032} C_VEL
LIN {X 0,Y 200.118,Z 559.558,A -85,B 0,C 180,E1 -21518.078,E2 -21518.078} C_VEL
LIN {X 0,Y 199.913,Z 559.57,A -85,B 0,C 180,E1 -21522.18,E2 -21522.18} C_VEL
LIN {X 0,Y 199.808,Z 559.595,A -85,B 0,C 180,E1 -21526.346,E2 -21526.346} C_VEL
LIN {X 0,Y 199.7,Z 559.593,A -85,B 0,C 180,E1 -21530.608,E2 -21530.608} C_VEL
LIN {X 0,Y 199.674,Z 559.601,A -85,B 0,C 180,E1 -21534.987,E2 -21534.987} C_VEL
LIN {X 0,Y 199.666,Z 559.614,A -85,B 0,C 180,E1 -21539.527,E2 -21539.527} C_VEL
LIN {X 0,Y 199.673,Z 559.604,A -85,B 0,C 180,E1 -21542.358,E2 -21542.358} C_VEL
LIN {X 0,Y 199.626,Z 559.62,A -85,B 0,C 180,E1 -21546.766,E2 -21546.766} C_VEL
LIN {X 0,Y 199.611,Z 559.614,A -85,B 0,C 180,E1 -21549.331,E2 -21549.331} C_VEL
LIN {X 0,Y 199.579,Z 559.618,A -85,B 0,C 180,E1 -21552.313,E2 -21552.313} C_VEL
LIN {X 0,Y 199.585,Z 559.625,A -85,B 0,C 180,E1 -21555.232,E2 -21555.232} C_VEL
LIN {X 0,Y 199.584,Z 559.618,A -85,B 0,C 180,E1 -21558.008,E2 -21558.008} C_VEL
LIN {X 0,Y 199.615,Z 559.604,A -85,B 0,C 180,E1 -21560.77,E2 -21560.77} C_VEL
LIN {X 0,Y 199.619,Z 559.62,A -85,B 0,C 180,E1 -21565.716,E2 -21565.716} C_VEL
LIN {X 0,Y 199.707,Z 559.604,A -85,B 0,C 180,E1 -21568.139,E2 -21568.139} C_VEL
LIN {X 0,Y 199.693,Z 559.598,A -85,B 0,C 180,E1 -21572.774,E2 -21572.774} C_VEL
LIN {X 0,Y 199.72,Z 559.606,A -85,B 0,C 180,E1 -21577.228,E2 -21577.228} C_VEL
LIN {X 0,Y 199.803,Z 559.581,A -85,B 0,C 180,E1 -21581.761,E2 -21581.761} C_VEL
LIN {X 0,Y 199.831,Z 559.589,A -85,B 0,C 180,E1 -21585.749,E2 -21585.749} C_VEL
LIN {X 0,Y 200.031,Z 559.566,A -85,B 0,C 180,E1 -21589.883,E2 -21589.883} C_VEL
LIN {X 0,Y 200.031,Z 559.555,A -85,B 0,C 180,E1 -21593.951,E2 -21593.951} C_VEL
LIN {X 0,Y 200.33,Z 559.532,A -85,B 0,C 180,E1 -21597.991,E2 -21597.991} C_VEL
LIN {X 0,Y 200.488,Z 559.51,A -85,B 0,C 180,E1 -21600.001,E2 -21600.001} C_VEL
LIN {X 0,Y 200.039,Z 559.556,A -85,B 0,C 180,E1 -21604.03,E2 -21604.03} C_VEL
LIN {X 0,Y 200.142,Z 559.556,A -85,B 0,C 180,E1 -21608.076,E2 -21608.076} C_VEL
LIN {X 0,Y 199.916,Z 559.573,A -85,B 0,C 180,E1 -21612.178,E2 -21612.178} C_VEL
LIN {X 0,Y 199.814,Z 559.597,A -85,B 0,C 180,E1 -21616.344,E2 -21616.344} C_VEL
LIN {X 0,Y 199.7,Z 559.6,A -85,B 0,C 180,E1 -21620.606,E2 -21620.606} C_VEL
LIN {X 0,Y 199.674,Z 559.588,A -85,B 0,C 180,E1 -21624.985,E2 -21624.985} C_VEL
LIN {X 0,Y 199.674,Z 559.612,A -85,B 0,C 180,E1 -21629.523,E2 -21629.523} C_VEL
LIN {X 0,Y 199.682,Z 559.609,A -85,B 0,C 180,E1 -21632.355,E2 -21632.355} C_VEL
LIN {X 0,Y 199.633,Z 559.619,A -85,B 0,C 180,E1 -21636.762,E2 -21636.762} C_VEL
LIN {X 0,Y 199.618,Z 559.619,A -85,B 0,C 180,E1 -21639.327,E2 -21639.327} C_VEL
LIN {X 0,Y 199.582,Z 559.624,A -85,B 0,C 180,E1 -21642.309,E2 -21642.309} C_VEL
LIN {X 0,Y 199.586,Z 559.617,A -85,B 0,C 180,E1 -21645.227,E2 -21645.227} C_VEL
LIN {X 0,Y 199.681,Z 559.75,A -85,B 0,C 180,E1 -21649.566,E2 -21649.566} C_VEL
LIN {X 0,Y 201.392,Z 566.893,A -85,B 0,C 180,E1 -21653.249,E2 -21653.249} C_VEL
LIN {X 0,Y 210.884,Z 590.863,A -85,B 0,C 180,E1 -21655.701,E2 -21655.701} C_VEL
LIN {X 0,Y 214.316,Z 600.289,A -85,B 0,C 180,E1 -21656.565,E2 -21656.565} C_VEL
LIN {X 0,Y 214.501,Z 601.791,A -85,B 0,C 180,E1 -21656.653,E2 -21656.653} C_VEL
LIN {X 0,Y 214.66,Z 607.627,A -85,B 0,C 180,E1 -21656.92,E2 -21656.92} C_VEL
LIN {X 0,Y 213.88,Z 613.512,A -85,B 0,C 180,E1 -21657.069,E2 -21657.069} C_VEL
LIN {X 0,Y 210.464,Z 629.226,A -85,B 0,C 180,E1 -21657.302,E2 -21657.302} C_VEL
LIN {X 0,Y 210,Z 633.206,A -85,B 0,C 180,E1 -21657.414,E2 -21657.414} C_VEL
LIN {X 0,Y 207.785,Z 675.688,A -85,B 0,C 180,E1 -21659.025,E2 -21659.025} C_VEL
LIN {X 0,Y 206.546,Z 688.046,A -85,B 0,C 180,E1 -21659.802,E2 -21659.802} C_VEL
LIN {X 0,Y 204.944,Z 699.952,A -85,B 0,C 180,E1 -21660.885,E2 -21660.885} C_VEL
LIN {X 0,Y 203.258,Z 710.506,A -85,B 0,C 180,E1 -21662.171,E2 -21662.171} C_VEL
LIN {X 0,Y 201.138,Z 721.196,A -85,B 0,C 180,E1 -21663.821,E2 -21663.821} C_VEL
LIN {X 0,Y 198.828,Z 732.187,A -85,B 0,C 180,E1 -21666.012,E2 -21666.012} C_VEL
LIN {X 0,Y 196.67,Z 741.619,A -85,B 0,C 180,E1 -21668.377,E2 -21668.377} C_VEL
LIN {X 0,Y 195.136,Z 748.653,A -85,B 0,C 180,E1 -21670.537,E2 -21670.537} C_VEL
LIN {X 0,Y 193.194,Z 756.851,A -85,B 0,C 180,E1 -21673.622,E2 -21673.622} C_VEL
LIN {X 0,Y 191.92,Z 762.388,A -85,B 0,C 180,E1 -21676.227,E2 -21676.227} C_VEL
LIN {X 0,Y 190.995,Z 767.797,A -85,B 0,C 180,E1 -21679.395,E2 -21679.395} C_VEL
LIN {X 0,Y 190.44,Z 771.965,A -85,B 0,C 180,E1 -21682.576,E2 -21682.576} C_VEL
LIN {X 0,Y 190.192,Z 775.327,A -85,B 0,C 180,E1 -21686.135,E2 -21686.135} C_VEL
LIN {X 0,Y 190.335,Z 777.524,A -85,B 0,C 180,E1 -21689.997,E2 -21689.997} C_VEL
LIN {X 0,Y 190.139,Z 778.313,A -85,B 0,C 180,E1 -21693.621,E2 -21693.621} C_VEL
LIN {X 0,Y 190.281,Z 778.157,A -85,B 0,C 180,E1 -21696.359,E2 -21696.359} C_VEL
LIN {X 0,Y 191.05,Z 776.544,A -85,B 0,C 180,E1 -21700.596,E2 -21700.596} C_VEL
LIN {X 0,Y 191.76,Z 775.155,A -85,B 0,C 180,E1 -21702.7,E2 -21702.7} C_VEL
LIN {X 0,Y 193.236,Z 772.265,A -85,B 0,C 180,E1 -21705.826,E2 -21705.826} C_VEL
LIN {X 0,Y 195.423,Z 768.385,A -85,B 0,C 180,E1 -21708.882,E2 -21708.882} C_VEL
LIN {X 0,Y 198.143,Z 763.41,A -85,B 0,C 180,E1 -21711.862,E2 -21711.862} C_VEL
LIN {X 0,Y 201.158,Z 757.212,A -85,B 0,C 180,E1 -21714.784,E2 -21714.784} C_VEL
LIN {X 0,Y 204.876,Z 749.543,A -85,B 0,C 180,E1 -21717.584,E2 -21717.584} C_VEL
LIN {X 0,Y 209.117,Z 739.979,A -85,B 0,C 180,E1 -21720.269,E2 -21720.269} C_VEL
LIN {X 0,Y 213.397,Z 729.182,A -85,B 0,C 180,E1 -21722.632,E2 -21722.632} C_VEL
LIN {X 0,Y 217.3,Z 718.05,A -85,B 0,C 180,E1 -21724.468,E2 -21724.468} C_VEL
LIN {X 0,Y 220.93,Z 705.605,A -85,B 0,C 180,E1 -21726.047,E2 -21726.047} C_VEL
LIN {X 0,Y 223.826,Z 693.273,A -85,B 0,C 180,E1 -21727.185,E2 -21727.185} C_VEL
LIN {X 0,Y 226.118,Z 680.576,A -85,B 0,C 180,E1 -21728.006,E2 -21728.006} C_VEL
LIN {X 0,Y 227.625,Z 666.669,A -85,B 0,C 180,E1 -21728.616,E2 -21728.616} C_VEL
LIN {X 0,Y 230.61,Z 627.068,A -85,B 0,C 180,E1 -21729.966,E2 -21729.966} C_VEL
LIN {X 0,Y 230.213,Z 624.189,A -85,B 0,C 180,E1 -21730.251,E2 -21730.251} C_VEL
LIN {X 0,Y 225.763,Z 613.208,A -85,B 0,C 180,E1 -21732.339,E2 -21732.339} C_VEL
LIN {X 0,Y 221.757,Z 604.679,A -85,B 0,C 180,E1 -21734.336,E2 -21734.336} C_VEL
LIN {X 0,Y 217.814,Z 597.538,A -85,B 0,C 180,E1 -21736.445,E2 -21736.445} C_VEL
LIN {X 0,Y 215.126,Z 592.938,A -85,B 0,C 180,E1 -21738.035,E2 -21738.035} C_VEL
LIN {X 0,Y 212.148,Z 588.05,A -85,B 0,C 180,E1 -21739.95,E2 -21739.95} C_VEL
LIN {X 0,Y 208.599,Z 582.589,A -85,B 0,C 180,E1 -21742.564,E2 -21742.564} C_VEL
LIN {X 0,Y 205.549,Z 578.212,A -85,B 0,C 180,E1 -21745.212,E2 -21745.212} C_VEL
LIN {X 0,Y 204.342,Z 576.459,A -85,B 0,C 180,E1 -21746.427,E2 -21746.427} C_VEL
LIN {X 0,Y 199.387,Z 569.428,A -85,B 0,C 180,E1 -21753.575,E2 -21753.575} C_VEL
LIN {X 0,Y 197.91,Z 567.907,A -85,B 0,C 180,E1 -21759.199,E2 -21759.199} C_VEL
LIN {X 0,Y 198.326,Z 567.801,A -85,B 0,C 180,E1 -21763.53,E2 -21763.53} C_VEL
LIN {X 0,Y 199.144,Z 568.278,A -85,B 0,C 180,E1 -21766.088,E2 -21766.088} C_VEL
LIN {X 0,Y 201.169,Z 570.954,A -85,B 0,C 180,E1 -21769.939,E2 -21769.939} C_VEL
LIN {X 0,Y 202.973,Z 572.581,A -85,B 0,C 180,E1 -21772.278,E2 -21772.278} C_VEL
LIN {X 0,Y 204.104,Z 573.85,A -85,B 0,C 180,E1 -21773.515,E2 -21773.515} C_VEL
LIN {X 0,Y 206.125,Z 576.579,A -85,B 0,C 180,E1 -21775.538,E2 -21775.538} C_VEL
LIN {X 0,Y 208.836,Z 579.113,A -85,B 0,C 180,E1 -21777.729,E2 -21777.729} C_VEL
LIN {X 0,Y 212.515,Z 584.551,A -85,B 0,C 180,E1 -21780.439,E2 -21780.439} C_VEL
LIN {X 0,Y 216.557,Z 590.609,A -85,B 0,C 180,E1 -21782.957,E2 -21782.957} C_VEL
LIN {X 0,Y 219.118,Z 594.672,A -85,B 0,C 180,E1 -21784.397,E2 -21784.397} C_VEL
LIN {X 0,Y 224.602,Z 604.61,A -85,B 0,C 180,E1 -21787.222,E2 -21787.222} C_VEL
LIN {X 0,Y 229.488,Z 614.853,A -85,B 0,C 180,E1 -21789.474,E2 -21789.474} C_VEL
LIN {X 0,Y 231.154,Z 619.063,A -85,B 0,C 180,E1 -21790.238,E2 -21790.238} C_VEL
LIN {X 0,Y 227.396,Z 666.081,A -85,B 0,C 180,E1 -21791.868,E2 -21791.868} C_VEL
LIN {X 0,Y 225.539,Z 679.063,A -85,B 0,C 180,E1 -21792.598,E2 -21792.598} C_VEL
LIN {X 0,Y 223.16,Z 691.361,A -85,B 0,C 180,E1 -21793.623,E2 -21793.623} C_VEL
LIN {X 0,Y 220.164,Z 703.209,A -85,B 0,C 180,E1 -21794.966,E2 -21794.966} C_VEL
LIN {X 0,Y 216.716,Z 714.35,A -85,B 0,C 180,E1 -21796.614,E2 -21796.614} C_VEL
LIN {X 0,Y 213.133,Z 724.504,A -85,B 0,C 180,E1 -21798.559,E2 -21798.559} C_VEL
LIN {X 0,Y 209.565,Z 733.116,A -85,B 0,C 180,E1 -21800.613,E2 -21800.613} C_VEL
LIN {X 0,Y 206.022,Z 740.882,A -85,B 0,C 180,E1 -21802.928,E2 -21802.928} C_VEL
LIN {X 0,Y 202.543,Z 747.899,A -85,B 0,C 180,E1 -21805.563,E2 -21805.563} C_VEL
LIN {X 0,Y 199.525,Z 753.622,A -85,B 0,C 180,E1 -21808.293,E2 -21808.293} C_VEL
LIN {X 0,Y 196.31,Z 759.149,A -85,B 0,C 180,E1 -21811.744,E2 -21811.744} C_VEL
LIN {X 0,Y 193.75,Z 763.388,A -85,B 0,C 180,E1 -21815.476,E2 -21815.476} C_VEL
LIN {X 0,Y 191.734,Z 766.325,A -85,B 0,C 180,E1 -21819.673,E2 -21819.673} C_VEL
LIN {X 0,Y 190.772,Z 767.399,A -85,B 0,C 180,E1 -21822.546,E2 -21822.546} C_VEL
LIN {X 0,Y 190.177,Z 767.736,A -85,B 0,C 180,E1 -21825.405,E2 -21825.405} C_VEL
LIN {X 0,Y 189.834,Z 767.323,A -85,B 0,C 180,E1 -21828.215,E2 -21828.215} C_VEL
LIN {X 0,Y 189.794,Z 766.225,A -85,B 0,C 180,E1 -21831.042,E2 -21831.042} C_VEL
LIN {X 0,Y 190.017,Z 763.907,A -85,B 0,C 180,E1 -21834.457,E2 -21834.457} C_VEL
LIN {X 0,Y 190.677,Z 760.321,A -85,B 0,C 180,E1 -21837.964,E2 -21837.964} C_VEL
LIN {X 0,Y 191.703,Z 755.143,A -85,B 0,C 180,E1 -21841.623,E2 -21841.623} C_VEL
LIN {X 0,Y 192.996,Z 749.264,A -85,B 0,C 180,E1 -21844.786,E2 -21844.786} C_VEL
LIN {X 0,Y 194.585,Z 742.37,A -85,B 0,C 180,E1 -21847.717,E2 -21847.717} C_VEL
LIN {X 0,Y 196.71,Z 733.515,A -85,B 0,C 180,E1 -21850.705,E2 -21850.705} C_VEL
LIN {X 0,Y 198.874,Z 724.06,A -85,B 0,C 180,E1 -21853.251,E2 -21853.251} C_VEL
LIN {X 0,Y 201.282,Z 712.919,A -85,B 0,C 180,E1 -21855.598,E2 -21855.598} C_VEL
LIN {X 0,Y 203.508,Z 700.898,A -85,B 0,C 180,E1 -21857.578,E2 -21857.578} C_VEL
LIN {X 0,Y 205.333,Z 689.318,A -85,B 0,C 180,E1 -21859.028,E2 -21859.028} C_VEL
LIN {X 0,Y 206.983,Z 675.617,A -85,B 0,C 180,E1 -21860.284,E2 -21860.284} C_VEL
LIN {X 0,Y 208.147,Z 662.393,A -85,B 0,C 180,E1 -21861.079,E2 -21861.079} C_VEL
LIN {X 0,Y 211.128,Z 603.708,A -85,B 0,C 180,E1 -21863.25,E2 -21863.25} C_VEL
LIN {X 0,Y 202.359,Z 579.799,A -85,B 0,C 180,E1 -21865.538,E2 -21865.538} C_VEL
LIN {X 0,Y 193.498,Z 561.642,A -85,B 0,C 180,E1 -21867.804,E2 -21867.804} C_VEL
LIN {X 0,Y 193.263,Z 560.411,A -85,B 0,C 180,E1 -21867.919,E2 -21867.919} C_VEL
LIN {X 0,Y 193.441,Z 560.389,A -85,B 0,C 180,E1 -21870.003,E2 -21870.003} C_VEL
LIN {X 0,Y 192.976,Z 560.443,A -85,B 0,C 180,E1 -21874.18,E2 -21874.18} C_VEL
LIN {X 0,Y 193.067,Z 560.437,A -85,B 0,C 180,E1 -21878.375,E2 -21878.375} C_VEL
LIN {X 0,Y 192.853,Z 560.447,A -85,B 0,C 180,E1 -21882.633,E2 -21882.633} C_VEL
LIN {X 0,Y 192.76,Z 560.475,A -85,B 0,C 180,E1 -21886.961,E2 -21886.961} C_VEL
LIN {X 0,Y 192.637,Z 560.465,A -85,B 0,C 180,E1 -21891.4,E2 -21891.4} C_VEL
LIN {X 0,Y 192.665,Z 560.471,A -85,B 0,C 180,E1 -21894.228,E2 -21894.228} C_VEL
LIN {X 0,Y 192.646,Z 560.49,A -85,B 0,C 180,E1 -21898.892,E2 -21898.892} C_VEL
LIN {X 0,Y 192.599,Z 560.487,A -85,B 0,C 180,E1 -21903.189,E2 -21903.189} C_VEL
LIN {X 0,Y 192.554,Z 560.497,A -85,B 0,C 180,E1 -21908.355,E2 -21908.355} C_VEL
LIN {X 0,Y 192.496,Z 560.503,A -85,B 0,C 180,E1 -21913.099,E2 -21913.099} C_VEL
LIN {X 0,Y 192.496,Z 560.506,A -85,B 0,C 180,E1 -21916.907,E2 -21916.907} C_VEL
LIN {X 0,Y 192.556,Z 560.488,A -85,B 0,C 180,E1 -21921.651,E2 -21921.651} C_VEL
LIN {X 0,Y 192.605,Z 560.492,A -85,B 0,C 180,E1 -21926.817,E2 -21926.817} C_VEL
LIN {X 0,Y 192.671,Z 560.469,A -85,B 0,C 180,E1 -21931.694,E2 -21931.694} C_VEL
LIN {X 0,Y 192.692,Z 560.481,A -85,B 0,C 180,E1 -21936.348,E2 -21936.348} C_VEL
LIN {X 0,Y 192.738,Z 560.462,A -85,B 0,C 180,E1 -21941.462,E2 -21941.462} C_VEL
LIN {X 0,Y 192.759,Z 560.466,A -85,B 0,C 180,E1 -21945.215,E2 -21945.215} C_VEL
LIN {X 0,Y 192.954,Z 560.449,A -85,B 0,C 180,E1 -21949.568,E2 -21949.568} C_VEL
LIN {X 0,Y 192.993,Z 560.43,A -85,B 0,C 180,E1 -21953.729,E2 -21953.729} C_VEL
LIN {X 0,Y 193.271,Z 560.411,A -85,B 0,C 180,E1 -21957.917,E2 -21957.917} C_VEL
LIN {X 0,Y 193.452,Z 560.387,A -85,B 0,C 180,E1 -21960.001,E2 -21960.001} C_VEL
LIN {X 0,Y 192.986,Z 560.434,A -85,B 0,C 180,E1 -21964.178,E2 -21964.178} C_VEL
LIN {X 0,Y 193.089,Z 560.433,A -85,B 0,C 180,E1 -21968.373,E2 -21968.373} C_VEL
LIN {X 0,Y 193.02,Z 560.438,A -85,B 0,C 180,E1 -21970.539,E2 -21970.539} C_VEL
LIN {X 0,Y 192.768,Z 560.473,A -85,B 0,C 180,E1 -21976.959,E2 -21976.959} C_VEL
LIN {X 0,Y 192.632,Z 560.475,A -85,B 0,C 180,E1 -21981.399,E2 -21981.399} C_VEL
LIN {X 0,Y 192.657,Z 560.456,A -85,B 0,C 180,E1 -21984.213,E2 -21984.213} C_VEL
LIN {X 0,Y 192.654,Z 560.486,A -85,B 0,C 180,E1 -21988.888,E2 -21988.888} C_VEL
LIN {X 0,Y 192.607,Z 560.492,A -85,B 0,C 180,E1 -21993.185,E2 -21993.185} C_VEL
LIN {X 0,Y 192.561,Z 560.501,A -85,B 0,C 180,E1 -21998.351,E2 -21998.351} C_VEL
LIN {X 0,Y 192.499,Z 560.506,A -85,B 0,C 180,E1 -22003.094,E2 -22003.094} C_VEL
LIN {X 0,Y 192.576,Z 560.553,A -85,B 0,C 180,E1 -22008.759,E2 -22008.759} C_VEL
LIN {X 0,Y 194.134,Z 566.866,A -85,B 0,C 180,E1 -22012.086,E2 -22012.086} C_VEL
LIN {X 0,Y 201.688,Z 585.307,A -85,B 0,C 180,E1 -22014.147,E2 -22014.147} C_VEL
LIN {X 0,Y 208.106,Z 602.587,A -85,B 0,C 180,E1 -22015.834,E2 -22015.834} C_VEL
LIN {X 0,Y 210.505,Z 622.987,A -85,B 0,C 180,E1 -22017.04,E2 -22017.04} C_VEL
LIN {X 0,Y 210,Z 633.206,A -85,B 0,C 180,E1 -22017.414,E2 -22017.414} C_VEL
LIN {X 0,Y 209.017,Z 639.028,A -85,B 0,C 180,E1 -22017.54,E2 -22017.54} C_VEL
LIN {X 0,Y 202.826,Z 657.883,A -85,B 0,C 180,E1 -22017.58,E2 -22017.58} C_VEL
LIN {X 0,Y 201.981,Z 663.7,A -85,B 0,C 180,E1 -22017.733,E2 -22017.733} C_VEL
LIN {X 0,Y 201.043,Z 679.217,A -85,B 0,C 180,E1 -22018.445,E2 -22018.445} C_VEL
LIN {X 0,Y 199.478,Z 692.419,A -85,B 0,C 180,E1 -22019.422,E2 -22019.422} C_VEL
LIN {X 0,Y 197.596,Z 704.625,A -85,B 0,C 180,E1 -22020.719,E2 -22020.719} C_VEL
LIN {X 0,Y 195.406,Z 716.534,A -85,B 0,C 180,E1 -22022.412,E2 -22022.412} C_VEL
LIN {X 0,Y 193.109,Z 727.236,A -85,B 0,C 180,E1 -22024.391,E2 -22024.391} C_VEL
LIN {X 0,Y 190.66,Z 737.934,A -85,B 0,C 180,E1 -22026.91,E2 -22026.91} C_VEL
LIN {X 0,Y 188.788,Z 745.999,A -85,B 0,C 180,E1 -22029.286,E2 -22029.286} C_VEL
LIN {X 0,Y 186.968,Z 753.361,A -85,B 0,C 180,E1 -22031.931,E2 -22031.931} C_VEL
LIN {X 0,Y 185.224,Z 760.563,A -85,B 0,C 180,E1 -22035.157,E2 -22035.157} C_VEL
LIN {X 0,Y 184,Z 767.115,A -85,B 0,C 180,E1 -22038.987,E2 -22038.987} C_VEL
LIN {X 0,Y 183.377,Z 771.391,A -85,B 0,C 180,E1 -22042.288,E2 -22042.288} C_VEL
LIN {X 0,Y 183.105,Z 775.141,A -85,B 0,C 180,E1 -22046.337,E2 -22046.337} C_VEL
LIN {X 0,Y 183.255,Z 777.201,A -85,B 0,C 180,E1 -22049.997,E2 -22049.997} C_VEL
LIN {X 0,Y 183.079,Z 778.112,A -85,B 0,C 180,E1 -22054.4,E2 -22054.4} C_VEL
LIN {X 0,Y 183.214,Z 777.985,A -85,B 0,C 180,E1 -22056.605,E2 -22056.605} C_VEL
LIN {X 0,Y 183.517,Z 777.449,A -85,B 0,C 180,E1 -22058.808,E2 -22058.808} C_VEL
LIN {X 0,Y 184.816,Z 775.166,A -85,B 0,C 180,E1 -22063.186,E2 -22063.186} C_VEL
LIN {X 0,Y 186.411,Z 772.392,A -85,B 0,C 180,E1 -22066.422,E2 -22066.422} C_VEL
LIN {X 0,Y 188.723,Z 768.622,A -85,B 0,C 180,E1 -22069.579,E2 -22069.579} C_VEL
LIN {X 0,Y 191.557,Z 763.764,A -85,B 0,C 180,E1 -22072.655,E2 -22072.655} C_VEL
LIN {X 0,Y 195.333,Z 756.584,A -85,B 0,C 180,E1 -22076.148,E2 -22076.148} C_VEL
LIN {X 0,Y 199.362,Z 748.827,A -85,B 0,C 180,E1 -22078.991,E2 -22078.991} C_VEL
LIN {X 0,Y 203.075,Z 740.976,A -85,B 0,C 180,E1 -22081.27,E2 -22081.27} C_VEL
LIN {X 0,Y 207.548,Z 730.42,A -85,B 0,C 180,E1 -22083.672,E2 -22083.672} C_VEL
LIN {X 0,Y 211.577,Z 719.722,A -85,B 0,C 180,E1 -22085.538,E2 -22085.538} C_VEL
LIN {X 0,Y 215.361,Z 707.697,A -85,B 0,C 180,E1 -22087.133,E2 -22087.133} C_VEL
LIN {X 0,Y 218.594,Z 695.115,A -85,B 0,C 180,E1 -22088.379,E2 -22088.379} C_VEL
LIN {X 0,Y 221.086,Z 682.532,A -85,B 0,C 180,E1 -22089.252,E2 -22089.252} C_VEL
LIN {X 0,Y 222.842,Z 668.47,A -85,B 0,C 180,E1 -22089.916,E2 -22089.916} C_VEL
LIN {X 0,Y 226.059,Z 628.136,A -85,B 0,C 180,E1 -22091.326,E2 -22091.326} C_VEL
LIN {X 0,Y 222.203,Z 618.19,A -85,B 0,C 180,E1 -22093.255,E2 -22093.255} C_VEL
LIN {X 0,Y 218.199,Z 609.273,A -85,B 0,C 180,E1 -22095.424,E2 -22095.424} C_VEL
LIN {X 0,Y 214.836,Z 603.02,A -85,B 0,C 180,E1 -22097.352,E2 -22097.352} C_VEL
LIN {X 0,Y 212.298,Z 598.489,A -85,B 0,C 180,E1 -22098.964,E2 -22098.964} C_VEL
LIN {X 0,Y 209.592,Z 593.861,A -85,B 0,C 180,E1 -22100.834,E2 -22100.834} C_VEL
LIN {X 0,Y 206.368,Z 588.74,A -85,B 0,C 180,E1 -22103.38,E2 -22103.38} C_VEL
LIN {X 0,Y 203.467,Z 584.151,A -85,B 0,C 180,E1 -22106.142,E2 -22106.142} C_VEL
LIN {X 0,Y 201.905,Z 582.252,A -85,B 0,C 180,E1 -22107.796,E2 -22107.796} C_VEL
LIN {X 0,Y 198.153,Z 576.307,A -85,B 0,C 180,E1 -22113.965,E2 -22113.965} C_VEL
LIN {X 0,Y 196.866,Z 574.932,A -85,B 0,C 180,E1 -22119.083,E2 -22119.083} C_VEL
LIN {X 0,Y 197.378,Z 574.862,A -85,B 0,C 180,E1 -22124.013,E2 -22124.013} C_VEL
LIN {X 0,Y 197.959,Z 575.289,A -85,B 0,C 180,E1 -22125.806,E2 -22125.806} C_VEL
LIN {X 0,Y 200.332,Z 578.215,A -85,B 0,C 180,E1 -22130.292,E2 -22130.292} C_VEL
LIN {X 0,Y 202.282,Z 580.184,A -85,B 0,C 180,E1 -22132.764,E2 -22132.764} C_VEL
LIN {X 0,Y 204.433,Z 583.251,A -85,B 0,C 180,E1 -22135.039,E2 -22135.039} C_VEL
LIN {X 0,Y 207.003,Z 585.801,A -85,B 0,C 180,E1 -22137.232,E2 -22137.232} C_VEL
LIN {X 0,Y 210.237,Z 590.764,A -85,B 0,C 180,E1 -22139.744,E2 -22139.744} C_VEL
LIN {X 0,Y 214.608,Z 597.603,A -85,B 0,C 180,E1 -22142.601,E2 -22142.601} C_VEL
LIN {X 0,Y 217.645,Z 603.016,A -85,B 0,C 180,E1 -22144.394,E2 -22144.394} C_VEL
LIN {X 0,Y 222.219,Z 611.775,A -85,B 0,C 180,E1 -22146.82,E2 -22146.82} C_VEL
LIN {X 0,Y 226.206,Z 620.838,A -85,B 0,C 180,E1 -22148.78,E2 -22148.78} C_VEL
LIN {X 0,Y 226.502,Z 621.613,A -85,B 0,C 180,E1 -22148.924,E2 -22148.924} C_VEL
LIN {X 0,Y 222.737,Z 666.43,A -85,B 0,C 180,E1 -22150.508,E2 -22150.508} C_VEL
LIN {X 0,Y 220.713,Z 679.809,A -85,B 0,C 180,E1 -22151.275,E2 -22151.275} C_VEL
LIN {X 0,Y 218.194,Z 692.049,A -85,B 0,C 180,E1 -22152.32,E2 -22152.32} C_VEL
LIN {X 0,Y 214.664,Z 705.064,A -85,B 0,C 180,E1 -22153.851,E2 -22153.851} C_VEL
LIN {X 0,Y 211.279,Z 715.377,A -85,B 0,C 180,E1 -22155.432,E2 -22155.432} C_VEL
LIN {X 0,Y 207.225,Z 726.092,A -85,B 0,C 180,E1 -22157.566,E2 -22157.566} C_VEL
LIN {X 0,Y 203.088,Z 735.34,A -85,B 0,C 180,E1 -22159.908,E2 -22159.908} C_VEL
LIN {X 0,Y 199.473,Z 742.664,A -85,B 0,C 180,E1 -22162.255,E2 -22162.255} C_VEL
LIN {X 0,Y 195.806,Z 749.489,A -85,B 0,C 180,E1 -22165.013,E2 -22165.013} C_VEL
LIN {X 0,Y 191.938,Z 756.104,A -85,B 0,C 180,E1 -22168.511,E2 -22168.511} C_VEL
LIN {X 0,Y 189.356,Z 760.222,A -85,B 0,C 180,E1 -22171.396,E2 -22171.396} C_VEL
LIN {X 0,Y 187.268,Z 763.382,A -85,B 0,C 180,E1 -22174.353,E2 -22174.353} C_VEL
LIN {X 0,Y 185.587,Z 765.653,A -85,B 0,C 180,E1 -22177.327,E2 -22177.327} C_VEL
LIN {X 0,Y 184.344,Z 767.158,A -85,B 0,C 180,E1 -22180.398,E2 -22180.398} C_VEL
LIN {X 0,Y 183.409,Z 767.89,A -85,B 0,C 180,E1 -22183.608,E2 -22183.608} C_VEL
LIN {X 0,Y 182.858,Z 767.761,A -85,B 0,C 180,E1 -22186.906,E2 -22186.906} C_VEL
LIN {X 0,Y 182.664,Z 766.676,A -85,B 0,C 180,E1 -22190.307,E2 -22190.307} C_VEL
LIN {X 0,Y 182.85,Z 764.529,A -85,B 0,C 180,E1 -22193.817,E2 -22193.817} C_VEL
LIN {X 0,Y 183.475,Z 760.976,A -85,B 0,C 180,E1 -22197.574,E2 -22197.574} C_VEL
LIN {X 0,Y 184.426,Z 756.169,A -85,B 0,C 180,E1 -22201.217,E2 -22201.217} C_VEL
LIN {X 0,Y 185.549,Z 751.31,A -85,B 0,C 180,E1 -22204.077,E2 -22204.077} C_VEL
LIN {X 0,Y 187.187,Z 744.289,A -85,B 0,C 180,E1 -22207.37,E2 -22207.37} C_VEL
LIN {X 0,Y 189.28,Z 735.885,A -85,B 0,C 180,E1 -22210.481,E2 -22210.481} C_VEL
LIN {X 0,Y 191.514,Z 726.547,A -85,B 0,C 180,E1 -22213.206,E2 -22213.206} C_VEL
LIN {X 0,Y 193.926,Z 715.948,A -85,B 0,C 180,E1 -22215.662,E2 -22215.662} C_VEL
LIN {X 0,Y 196.052,Z 705.476,A -85,B 0,C 180,E1 -22217.583,E2 -22217.583} C_VEL
LIN {X 0,Y 198.045,Z 693.679,A -85,B 0,C 180,E1 -22219.266,E2 -22219.266} C_VEL
LIN {X 0,Y 199.78,Z 681.729,A -85,B 0,C 180,E1 -22220.545,E2 -22220.545} C_VEL
LIN {X 0,Y 201.163,Z 668.521,A -85,B 0,C 180,E1 -22221.552,E2 -22221.552} C_VEL
LIN {X 0,Y 202.248,Z 651.826,A -85,B 0,C 180,E1 -22222.3,E2 -22222.3} C_VEL
LIN {X 0,Y 204.711,Z 605.429,A -85,B 0,C 180,E1 -22224.042,E2 -22224.042} C_VEL
LIN {X 0,Y 196.522,Z 582.856,A -85,B 0,C 180,E1 -22226.287,E2 -22226.287} C_VEL
LIN {X 0,Y 186.394,Z 561.945,A -85,B 0,C 180,E1 -22229.025,E2 -22229.025} C_VEL
LIN {X 0,Y 186.3,Z 561.282,A -85,B 0,C 180,E1 -22229.193,E2 -22229.193} C_VEL
LIN {X 0,Y 186.206,Z 561.289,A -85,B 0,C 180,E1 -22232.166,E2 -22232.166} C_VEL
LIN {X 0,Y 186.012,Z 561.317,A -85,B 0,C 180,E1 -22238.695,E2 -22238.695} C_VEL
LIN {X 0,Y 185.764,Z 561.329,A -85,B 0,C 180,E1 -22243.123,E2 -22243.123} C_VEL
LIN {X 0,Y 185.692,Z 561.354,A -85,B 0,C 180,E1 -22247.628,E2 -22247.628} C_VEL
LIN {X 0,Y 185.597,Z 561.337,A -85,B 0,C 180,E1 -22252.254,E2 -22252.254} C_VEL
LIN {X 0,Y 185.562,Z 561.369,A -85,B 0,C 180,E1 -22257.035,E2 -22257.035} C_VEL
LIN {X 0,Y 185.579,Z 561.369,A -85,B 0,C 180,E1 -22259.496,E2 -22259.496} C_VEL
LIN {X 0,Y 185.501,Z 561.376,A -85,B 0,C 180,E1 -22264.635,E2 -22264.635} C_VEL
LIN {X 0,Y 185.509,Z 561.378,A -85,B 0,C 180,E1 -22267.316,E2 -22267.316} C_VEL
LIN {X 0,Y 185.475,Z 561.37,A -85,B 0,C 180,E1 -22270.728,E2 -22270.728} C_VEL
LIN {X 0,Y 185.483,Z 561.38,A -85,B 0,C 180,E1 -22273.954,E2 -22273.954} C_VEL
LIN {X 0,Y 185.476,Z 561.369,A -85,B 0,C 180,E1 -22279.278,E2 -22279.278} C_VEL
LIN {X 0,Y 185.511,Z 561.369,A -85,B 0,C 180,E1 -22282.714,E2 -22282.714} C_VEL
LIN {X 0,Y 185.552,Z 561.367,A -85,B 0,C 180,E1 -22287.978,E2 -22287.978} C_VEL
LIN {X 0,Y 185.588,Z 561.352,A -85,B 0,C 180,E1 -22290.578,E2 -22290.578} C_VEL
LIN {X 0,Y 185.587,Z 561.365,A -85,B 0,C 180,E1 -22295.384,E2 -22295.384} C_VEL
LIN {X 0,Y 185.665,Z 561.345,A -85,B 0,C 180,E1 -22301.151,E2 -22301.151} C_VEL
LIN {X 0,Y 185.692,Z 561.345,A -85,B 0,C 180,E1 -22304.638,E2 -22304.638} C_VEL
LIN {X 0,Y 185.897,Z 561.328,A -85,B 0,C 180,E1 -22309.419,E2 -22309.419} C_VEL
LIN {X 0,Y 185.956,Z 561.306,A -85,B 0,C 180,E1 -22313.491,E2 -22313.491} C_VEL
LIN {X 0,Y 186.215,Z 561.289,A -85,B 0,C 180,E1 -22317.838,E2 -22317.838} C_VEL
LIN {X 0,Y 186.416,Z 561.263,A -85,B 0,C 180,E1 -22320.001,E2 -22320.001} C_VEL
LIN {X 0,Y 185.934,Z 561.312,A -85,B 0,C 180,E1 -22324.337,E2 -22324.337} C_VEL
LIN {X 0,Y 186.039,Z 561.311,A -85,B 0,C 180,E1 -22328.692,E2 -22328.692} C_VEL
LIN {X 0,Y 185.752,Z 561.335,A -85,B 0,C 180,E1 -22333.122,E2 -22333.122} C_VEL
LIN {X 0,Y 185.7,Z 561.355,A -85,B 0,C 180,E1 -22337.625,E2 -22337.625} C_VEL
LIN {X 0,Y 185.591,Z 561.343,A -85,B 0,C 180,E1 -22342.253,E2 -22342.253} C_VEL
